// TIA Portal V16 export
// export: Created 2024-09-05T17:39:23.0698043Z, ExportSetting WithDefaults, DisplayName Totally Integrated Automation Portal, DisplayVersion V16 Update 6, DisplayName TIA Portal Version Control Interface, DisplayVersion V16 Update 2, DisplayName TIA Portal Openness, DisplayVersion V16 Update 6, DisplayName STEP 7 Professional, DisplayVersion V16 Update 6, DisplayName STEP 7 Safety, DisplayVersion V16, DisplayName WinCC Advanced, DisplayVersion V16 Update 6
FUNCTION "FC_CONFIG_MSG_IJC" : Void   // FC2, LAD
{ S7_Optimized_Access := 'TRUE' }
VERSION : 0.1
// stored: AutoNumber true, IsIECCheckEnabled false, SetENOAutomatically false, UDAEnableTagReadback false
   VAR_TEMP
      STRING_USER1 : String;
      STRING_USER2 : String;
      STRING_CORDON_1 : String;
      INDEX_IJC_CORDON : Int;
      STRING_CORDONES : Array[0..13] of String;
   END_VAR
   VAR_TEMP   // added for the SCL form of the ladder/FBD networks
      _w1 : Bool;
      _w2 : Bool;
   END_VAR
BEGIN

REGION Network 1: INDEX MSG CONFIG
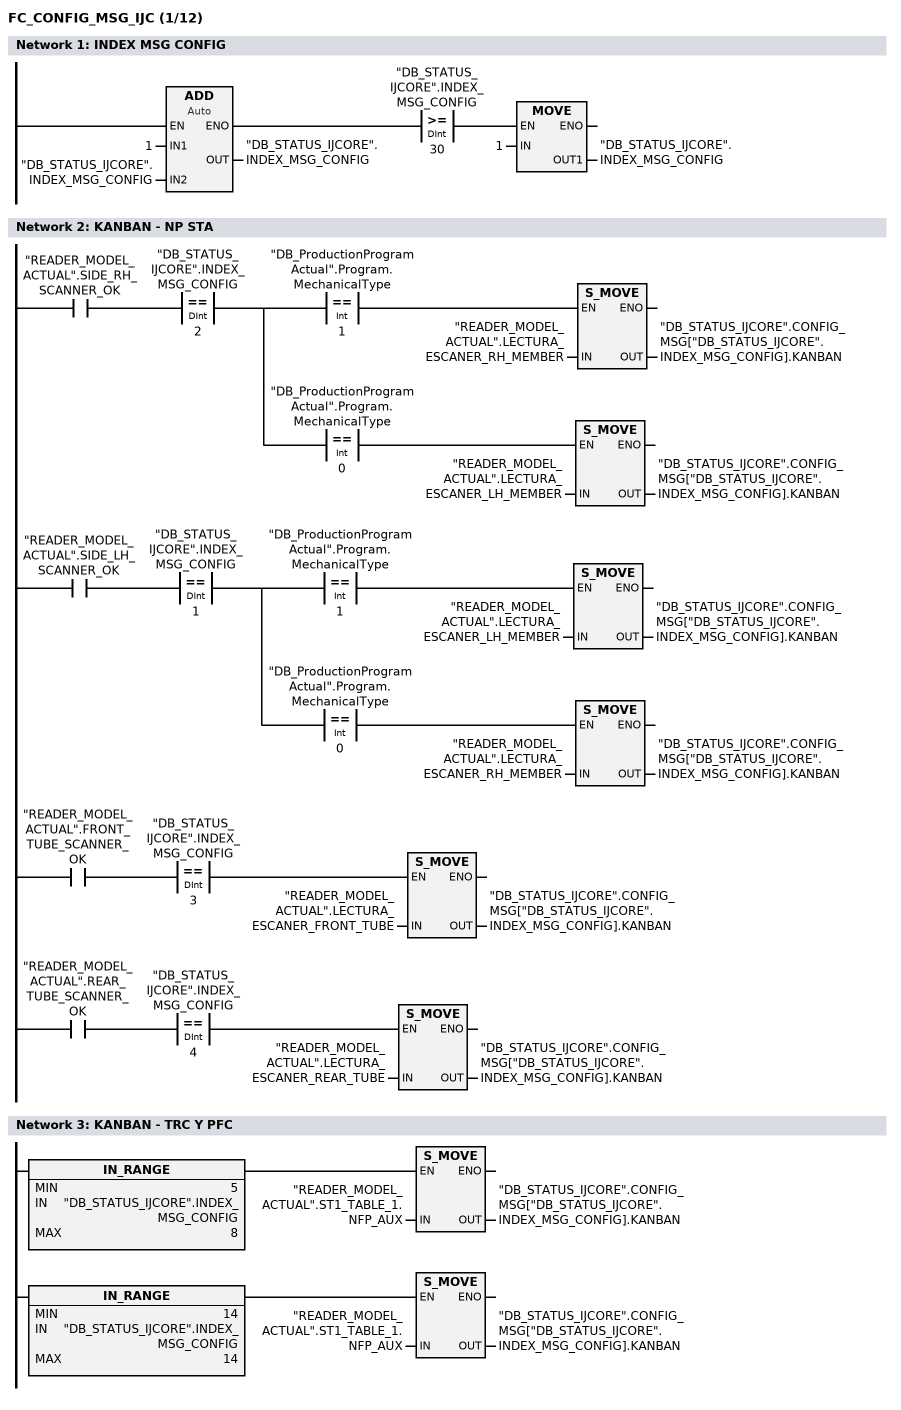
   RUNG wire#powerrail
      Add(in1 := 1, in2 := "DB_STATUS_IJCORE".INDEX_MSG_CONFIG, out => "DB_STATUS_IJCORE".INDEX_MSG_CONFIG)
      { S7_Templates := "SrcType := DInt" } GE_Contact(in1 := "DB_STATUS_IJCORE".INDEX_MSG_CONFIG, in2 := 30)
      Move(in := 1, out1 => "DB_STATUS_IJCORE".INDEX_MSG_CONFIG)
   END_RUNG
   // the same network as SCL:
   "DB_STATUS_IJCORE".INDEX_MSG_CONFIG := 1 + "DB_STATUS_IJCORE".INDEX_MSG_CONFIG;
   IF "DB_STATUS_IJCORE".INDEX_MSG_CONFIG >= 30 THEN "DB_STATUS_IJCORE".INDEX_MSG_CONFIG := 1; END_IF;
END_REGION

REGION Network 2: KANBAN - NP STA
   RUNG wire#powerrail
      Contact( "READER_MODEL_ACTUAL".SIDE_RH_SCANNER_OK )
      { S7_Templates := "SrcType := DInt" } EQ_Contact(in1 := "DB_STATUS_IJCORE".INDEX_MSG_CONFIG, in2 := 2)
      wire#w1
      { S7_Templates := "SrcType := Int" } EQ_Contact(in1 := "DB_ProductionProgramActual".Program.MechanicalType, in2 := 1)
      S_Move(in := "READER_MODEL_ACTUAL".LECTURA_ESCANER_RH_MEMBER, out => "DB_STATUS_IJCORE".CONFIG_MSG["DB_STATUS_IJCORE".INDEX_MSG_CONFIG].KANBAN)
   END_RUNG
   RUNG wire#w1
      { S7_Templates := "SrcType := Int" } EQ_Contact(in1 := "DB_ProductionProgramActual".Program.MechanicalType, in2 := 0)
      S_Move(in := "READER_MODEL_ACTUAL".LECTURA_ESCANER_LH_MEMBER, out => "DB_STATUS_IJCORE".CONFIG_MSG["DB_STATUS_IJCORE".INDEX_MSG_CONFIG].KANBAN)
   END_RUNG
   RUNG wire#powerrail
      Contact( "READER_MODEL_ACTUAL".SIDE_LH_SCANNER_OK )
      { S7_Templates := "SrcType := DInt" } EQ_Contact(in1 := "DB_STATUS_IJCORE".INDEX_MSG_CONFIG, in2 := 1)
      wire#w2
      { S7_Templates := "SrcType := Int" } EQ_Contact(in1 := "DB_ProductionProgramActual".Program.MechanicalType, in2 := 1)
      S_Move(in := "READER_MODEL_ACTUAL".LECTURA_ESCANER_LH_MEMBER, out => "DB_STATUS_IJCORE".CONFIG_MSG["DB_STATUS_IJCORE".INDEX_MSG_CONFIG].KANBAN)
   END_RUNG
   RUNG wire#w2
      { S7_Templates := "SrcType := Int" } EQ_Contact(in1 := "DB_ProductionProgramActual".Program.MechanicalType, in2 := 0)
      S_Move(in := "READER_MODEL_ACTUAL".LECTURA_ESCANER_RH_MEMBER, out => "DB_STATUS_IJCORE".CONFIG_MSG["DB_STATUS_IJCORE".INDEX_MSG_CONFIG].KANBAN)
   END_RUNG
   RUNG wire#powerrail
      Contact( "READER_MODEL_ACTUAL".FRONT_TUBE_SCANNER_OK )
      { S7_Templates := "SrcType := DInt" } EQ_Contact(in1 := "DB_STATUS_IJCORE".INDEX_MSG_CONFIG, in2 := 3)
      S_Move(in := "READER_MODEL_ACTUAL".LECTURA_ESCANER_FRONT_TUBE, out => "DB_STATUS_IJCORE".CONFIG_MSG["DB_STATUS_IJCORE".INDEX_MSG_CONFIG].KANBAN)
   END_RUNG
   RUNG wire#powerrail
      Contact( "READER_MODEL_ACTUAL".REAR_TUBE_SCANNER_OK )
      { S7_Templates := "SrcType := DInt" } EQ_Contact(in1 := "DB_STATUS_IJCORE".INDEX_MSG_CONFIG, in2 := 4)
      S_Move(in := "READER_MODEL_ACTUAL".LECTURA_ESCANER_REAR_TUBE, out => "DB_STATUS_IJCORE".CONFIG_MSG["DB_STATUS_IJCORE".INDEX_MSG_CONFIG].KANBAN)
   END_RUNG
   // the same network as SCL:
   #_w1 := "READER_MODEL_ACTUAL".SIDE_RH_SCANNER_OK AND ("DB_STATUS_IJCORE".INDEX_MSG_CONFIG = 2);
   IF #_w1 AND ("DB_ProductionProgramActual".Program.MechanicalType = 1) THEN
       "DB_STATUS_IJCORE".CONFIG_MSG["DB_STATUS_IJCORE".INDEX_MSG_CONFIG].KANBAN := "READER_MODEL_ACTUAL".LECTURA_ESCANER_RH_MEMBER;
   END_IF;
   IF #_w1 AND ("DB_ProductionProgramActual".Program.MechanicalType = 0) THEN
       "DB_STATUS_IJCORE".CONFIG_MSG["DB_STATUS_IJCORE".INDEX_MSG_CONFIG].KANBAN := "READER_MODEL_ACTUAL".LECTURA_ESCANER_LH_MEMBER;
   END_IF;
   #_w2 := "READER_MODEL_ACTUAL".SIDE_LH_SCANNER_OK AND ("DB_STATUS_IJCORE".INDEX_MSG_CONFIG = 1);
   IF #_w2 AND ("DB_ProductionProgramActual".Program.MechanicalType = 1) THEN
       "DB_STATUS_IJCORE".CONFIG_MSG["DB_STATUS_IJCORE".INDEX_MSG_CONFIG].KANBAN := "READER_MODEL_ACTUAL".LECTURA_ESCANER_LH_MEMBER;
   END_IF;
   IF #_w2 AND ("DB_ProductionProgramActual".Program.MechanicalType = 0) THEN
       "DB_STATUS_IJCORE".CONFIG_MSG["DB_STATUS_IJCORE".INDEX_MSG_CONFIG].KANBAN := "READER_MODEL_ACTUAL".LECTURA_ESCANER_RH_MEMBER;
   END_IF;
   IF "READER_MODEL_ACTUAL".FRONT_TUBE_SCANNER_OK AND ("DB_STATUS_IJCORE".INDEX_MSG_CONFIG = 3) THEN
       "DB_STATUS_IJCORE".CONFIG_MSG["DB_STATUS_IJCORE".INDEX_MSG_CONFIG].KANBAN := "READER_MODEL_ACTUAL".LECTURA_ESCANER_FRONT_TUBE;
   END_IF;
   IF "READER_MODEL_ACTUAL".REAR_TUBE_SCANNER_OK AND ("DB_STATUS_IJCORE".INDEX_MSG_CONFIG = 4) THEN
       "DB_STATUS_IJCORE".CONFIG_MSG["DB_STATUS_IJCORE".INDEX_MSG_CONFIG].KANBAN := "READER_MODEL_ACTUAL".LECTURA_ESCANER_REAR_TUBE;
   END_IF;
END_REGION

REGION Network 3: KANBAN - TRC Y PFC
   RUNG wire#powerrail
      { S7_Templates := "SrcType := DInt" } InRange(min := 5, in := "DB_STATUS_IJCORE".INDEX_MSG_CONFIG, max := 8)
      S_Move(in := "READER_MODEL_ACTUAL".ST1_TABLE_1.NFP_AUX, out => "DB_STATUS_IJCORE".CONFIG_MSG["DB_STATUS_IJCORE".INDEX_MSG_CONFIG].KANBAN)
   END_RUNG
   RUNG wire#powerrail
      { S7_Templates := "SrcType := DInt" } InRange(min := 14, in := "DB_STATUS_IJCORE".INDEX_MSG_CONFIG, max := 14)
      S_Move(in := "READER_MODEL_ACTUAL".ST1_TABLE_1.NFP_AUX, out => "DB_STATUS_IJCORE".CONFIG_MSG["DB_STATUS_IJCORE".INDEX_MSG_CONFIG].KANBAN)
   END_RUNG
   // the same network as SCL:
   IF (5 <= "DB_STATUS_IJCORE".INDEX_MSG_CONFIG) AND ("DB_STATUS_IJCORE".INDEX_MSG_CONFIG <= 8) THEN
       "DB_STATUS_IJCORE".CONFIG_MSG["DB_STATUS_IJCORE".INDEX_MSG_CONFIG].KANBAN := "READER_MODEL_ACTUAL".ST1_TABLE_1.NFP_AUX;
   END_IF;
   IF (14 <= "DB_STATUS_IJCORE".INDEX_MSG_CONFIG) AND ("DB_STATUS_IJCORE".INDEX_MSG_CONFIG <= 14) THEN
       "DB_STATUS_IJCORE".CONFIG_MSG["DB_STATUS_IJCORE".INDEX_MSG_CONFIG].KANBAN := "READER_MODEL_ACTUAL".ST1_TABLE_1.NFP_AUX;
   END_IF;
END_REGION

REGION Network 4: KANBAN - TRR Y CNF
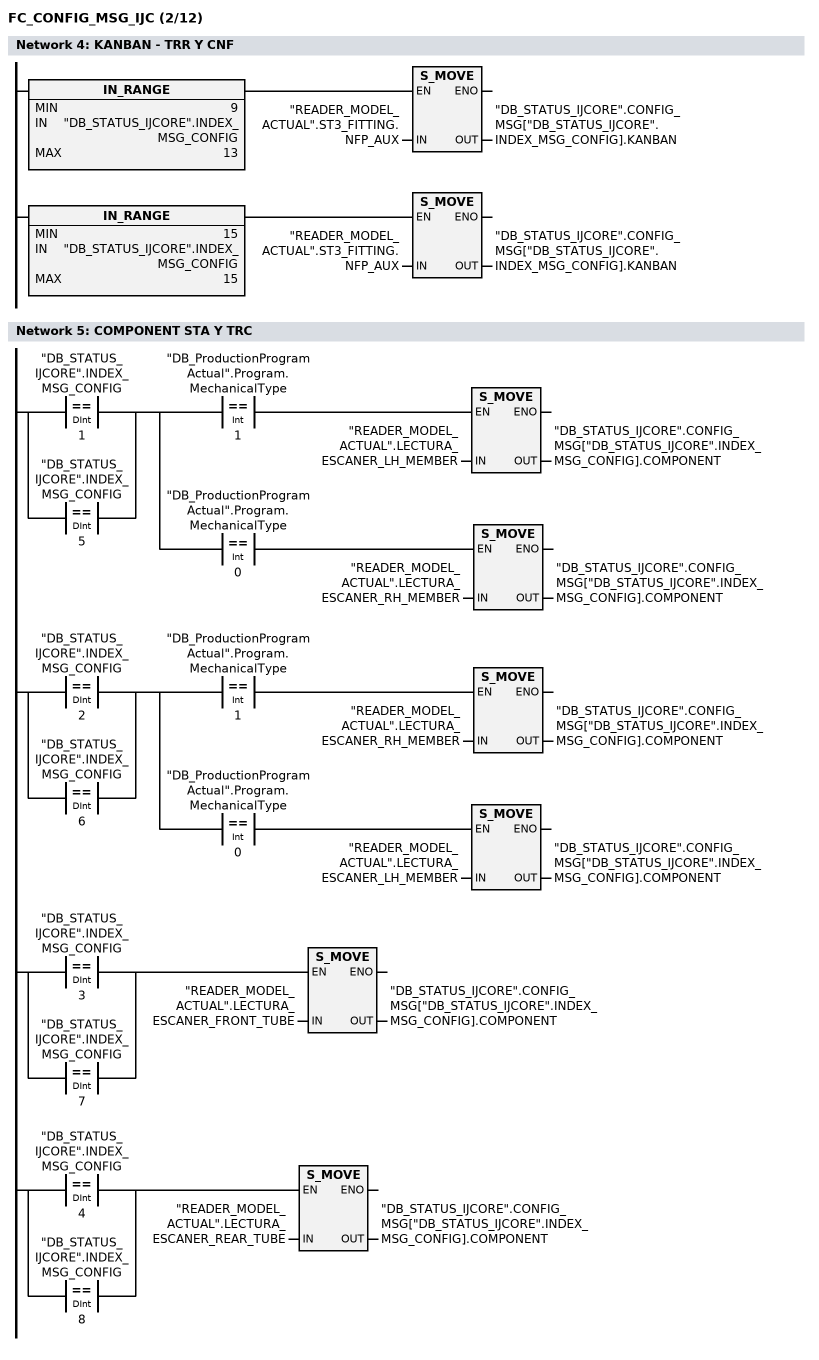
   RUNG wire#powerrail
      { S7_Templates := "SrcType := DInt" } InRange(min := 9, in := "DB_STATUS_IJCORE".INDEX_MSG_CONFIG, max := 13)
      S_Move(in := "READER_MODEL_ACTUAL".ST3_FITTING.NFP_AUX, out => "DB_STATUS_IJCORE".CONFIG_MSG["DB_STATUS_IJCORE".INDEX_MSG_CONFIG].KANBAN)
   END_RUNG
   RUNG wire#powerrail
      { S7_Templates := "SrcType := DInt" } InRange(min := 15, in := "DB_STATUS_IJCORE".INDEX_MSG_CONFIG, max := 15)
      S_Move(in := "READER_MODEL_ACTUAL".ST3_FITTING.NFP_AUX, out => "DB_STATUS_IJCORE".CONFIG_MSG["DB_STATUS_IJCORE".INDEX_MSG_CONFIG].KANBAN)
   END_RUNG
   // the same network as SCL:
   IF (9 <= "DB_STATUS_IJCORE".INDEX_MSG_CONFIG) AND ("DB_STATUS_IJCORE".INDEX_MSG_CONFIG <= 13) THEN
       "DB_STATUS_IJCORE".CONFIG_MSG["DB_STATUS_IJCORE".INDEX_MSG_CONFIG].KANBAN := "READER_MODEL_ACTUAL".ST3_FITTING.NFP_AUX;
   END_IF;
   IF (15 <= "DB_STATUS_IJCORE".INDEX_MSG_CONFIG) AND ("DB_STATUS_IJCORE".INDEX_MSG_CONFIG <= 15) THEN
       "DB_STATUS_IJCORE".CONFIG_MSG["DB_STATUS_IJCORE".INDEX_MSG_CONFIG].KANBAN := "READER_MODEL_ACTUAL".ST3_FITTING.NFP_AUX;
   END_IF;
END_REGION

REGION Network 5: COMPONENT STA Y TRC
   RUNG wire#powerrail
      { S7_Templates := "SrcType := DInt" } EQ_Contact(in1 := "DB_STATUS_IJCORE".INDEX_MSG_CONFIG, in2 := 1)
      wire#w1
      { S7_Templates := "SrcType := Int" } EQ_Contact(in1 := "DB_ProductionProgramActual".Program.MechanicalType, in2 := 1)
      S_Move(in := "READER_MODEL_ACTUAL".LECTURA_ESCANER_LH_MEMBER, out => "DB_STATUS_IJCORE".CONFIG_MSG["DB_STATUS_IJCORE".INDEX_MSG_CONFIG].COMPONENT)
   END_RUNG
   RUNG wire#powerrail
      { S7_Templates := "SrcType := DInt" } EQ_Contact(in1 := "DB_STATUS_IJCORE".INDEX_MSG_CONFIG, in2 := 5)
   END_RUNG wire#w1
   RUNG wire#w1
      { S7_Templates := "SrcType := Int" } EQ_Contact(in1 := "DB_ProductionProgramActual".Program.MechanicalType, in2 := 0)
      S_Move(in := "READER_MODEL_ACTUAL".LECTURA_ESCANER_RH_MEMBER, out => "DB_STATUS_IJCORE".CONFIG_MSG["DB_STATUS_IJCORE".INDEX_MSG_CONFIG].COMPONENT)
   END_RUNG
   RUNG wire#powerrail
      { S7_Templates := "SrcType := DInt" } EQ_Contact(in1 := "DB_STATUS_IJCORE".INDEX_MSG_CONFIG, in2 := 2)
      wire#w2
      { S7_Templates := "SrcType := Int" } EQ_Contact(in1 := "DB_ProductionProgramActual".Program.MechanicalType, in2 := 1)
      S_Move(in := "READER_MODEL_ACTUAL".LECTURA_ESCANER_RH_MEMBER, out => "DB_STATUS_IJCORE".CONFIG_MSG["DB_STATUS_IJCORE".INDEX_MSG_CONFIG].COMPONENT)
   END_RUNG
   RUNG wire#powerrail
      { S7_Templates := "SrcType := DInt" } EQ_Contact(in1 := "DB_STATUS_IJCORE".INDEX_MSG_CONFIG, in2 := 6)
   END_RUNG wire#w2
   RUNG wire#w2
      { S7_Templates := "SrcType := Int" } EQ_Contact(in1 := "DB_ProductionProgramActual".Program.MechanicalType, in2 := 0)
      S_Move(in := "READER_MODEL_ACTUAL".LECTURA_ESCANER_LH_MEMBER, out => "DB_STATUS_IJCORE".CONFIG_MSG["DB_STATUS_IJCORE".INDEX_MSG_CONFIG].COMPONENT)
   END_RUNG
   RUNG wire#powerrail
      { S7_Templates := "SrcType := DInt" } EQ_Contact(in1 := "DB_STATUS_IJCORE".INDEX_MSG_CONFIG, in2 := 3)
      wire#w3
      S_Move(in := "READER_MODEL_ACTUAL".LECTURA_ESCANER_FRONT_TUBE, out => "DB_STATUS_IJCORE".CONFIG_MSG["DB_STATUS_IJCORE".INDEX_MSG_CONFIG].COMPONENT)
   END_RUNG
   RUNG wire#powerrail
      { S7_Templates := "SrcType := DInt" } EQ_Contact(in1 := "DB_STATUS_IJCORE".INDEX_MSG_CONFIG, in2 := 7)
   END_RUNG wire#w3
   RUNG wire#powerrail
      { S7_Templates := "SrcType := DInt" } EQ_Contact(in1 := "DB_STATUS_IJCORE".INDEX_MSG_CONFIG, in2 := 4)
      wire#w4
      S_Move(in := "READER_MODEL_ACTUAL".LECTURA_ESCANER_REAR_TUBE, out => "DB_STATUS_IJCORE".CONFIG_MSG["DB_STATUS_IJCORE".INDEX_MSG_CONFIG].COMPONENT)
   END_RUNG
   RUNG wire#powerrail
      { S7_Templates := "SrcType := DInt" } EQ_Contact(in1 := "DB_STATUS_IJCORE".INDEX_MSG_CONFIG, in2 := 8)
   END_RUNG wire#w4
   // the same network as SCL:
   #_w1 := ("DB_STATUS_IJCORE".INDEX_MSG_CONFIG = 1) OR ("DB_STATUS_IJCORE".INDEX_MSG_CONFIG = 5);
   IF #_w1 AND ("DB_ProductionProgramActual".Program.MechanicalType = 1) THEN
       "DB_STATUS_IJCORE".CONFIG_MSG["DB_STATUS_IJCORE".INDEX_MSG_CONFIG].COMPONENT := "READER_MODEL_ACTUAL".LECTURA_ESCANER_LH_MEMBER;
   END_IF;
   IF #_w1 AND ("DB_ProductionProgramActual".Program.MechanicalType = 0) THEN
       "DB_STATUS_IJCORE".CONFIG_MSG["DB_STATUS_IJCORE".INDEX_MSG_CONFIG].COMPONENT := "READER_MODEL_ACTUAL".LECTURA_ESCANER_RH_MEMBER;
   END_IF;
   #_w2 := ("DB_STATUS_IJCORE".INDEX_MSG_CONFIG = 2) OR ("DB_STATUS_IJCORE".INDEX_MSG_CONFIG = 6);
   IF #_w2 AND ("DB_ProductionProgramActual".Program.MechanicalType = 1) THEN
       "DB_STATUS_IJCORE".CONFIG_MSG["DB_STATUS_IJCORE".INDEX_MSG_CONFIG].COMPONENT := "READER_MODEL_ACTUAL".LECTURA_ESCANER_RH_MEMBER;
   END_IF;
   IF #_w2 AND ("DB_ProductionProgramActual".Program.MechanicalType = 0) THEN
       "DB_STATUS_IJCORE".CONFIG_MSG["DB_STATUS_IJCORE".INDEX_MSG_CONFIG].COMPONENT := "READER_MODEL_ACTUAL".LECTURA_ESCANER_LH_MEMBER;
   END_IF;
   IF ("DB_STATUS_IJCORE".INDEX_MSG_CONFIG = 3) OR ("DB_STATUS_IJCORE".INDEX_MSG_CONFIG = 7) THEN
       "DB_STATUS_IJCORE".CONFIG_MSG["DB_STATUS_IJCORE".INDEX_MSG_CONFIG].COMPONENT := "READER_MODEL_ACTUAL".LECTURA_ESCANER_FRONT_TUBE;
   END_IF;
   IF ("DB_STATUS_IJCORE".INDEX_MSG_CONFIG = 4) OR ("DB_STATUS_IJCORE".INDEX_MSG_CONFIG = 8) THEN
       "DB_STATUS_IJCORE".CONFIG_MSG["DB_STATUS_IJCORE".INDEX_MSG_CONFIG].COMPONENT := "READER_MODEL_ACTUAL".LECTURA_ESCANER_REAR_TUBE;
   END_IF;
END_REGION

REGION Network 6: COMPONENT PFC
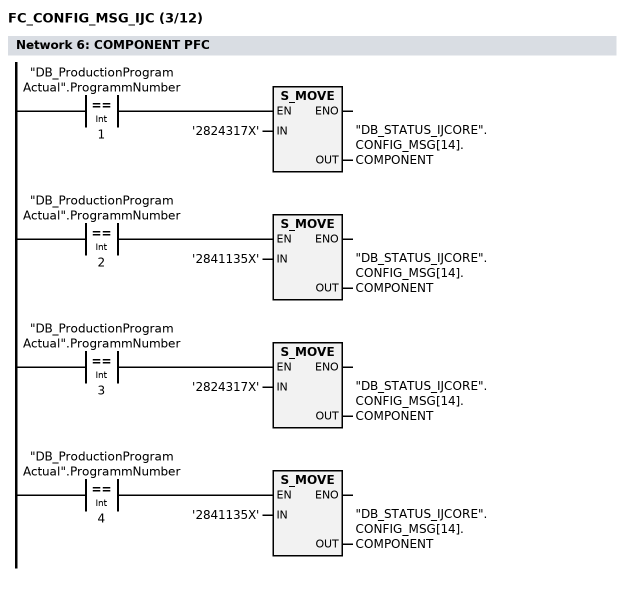
   RUNG wire#powerrail
      { S7_Templates := "SrcType := Int" } EQ_Contact(in1 := "DB_ProductionProgramActual".ProgrammNumber, in2 := 1)
      S_Move(in := '2824317X', out => "DB_STATUS_IJCORE".CONFIG_MSG[14].COMPONENT)
   END_RUNG
   RUNG wire#powerrail
      { S7_Templates := "SrcType := Int" } EQ_Contact(in1 := "DB_ProductionProgramActual".ProgrammNumber, in2 := 2)
      S_Move(in := '2841135X', out => "DB_STATUS_IJCORE".CONFIG_MSG[14].COMPONENT)
   END_RUNG
   RUNG wire#powerrail
      { S7_Templates := "SrcType := Int" } EQ_Contact(in1 := "DB_ProductionProgramActual".ProgrammNumber, in2 := 3)
      S_Move(in := '2824317X', out => "DB_STATUS_IJCORE".CONFIG_MSG[14].COMPONENT)
   END_RUNG
   RUNG wire#powerrail
      { S7_Templates := "SrcType := Int" } EQ_Contact(in1 := "DB_ProductionProgramActual".ProgrammNumber, in2 := 4)
      S_Move(in := '2841135X', out => "DB_STATUS_IJCORE".CONFIG_MSG[14].COMPONENT)
   END_RUNG
   // the same network as SCL:
   IF "DB_ProductionProgramActual".ProgrammNumber = 1 THEN
       "DB_STATUS_IJCORE".CONFIG_MSG[14].COMPONENT := '2824317X';
   END_IF;
   IF "DB_ProductionProgramActual".ProgrammNumber = 2 THEN
       "DB_STATUS_IJCORE".CONFIG_MSG[14].COMPONENT := '2841135X';
   END_IF;
   IF "DB_ProductionProgramActual".ProgrammNumber = 3 THEN
       "DB_STATUS_IJCORE".CONFIG_MSG[14].COMPONENT := '2824317X';
   END_IF;
   IF "DB_ProductionProgramActual".ProgrammNumber = 4 THEN
       "DB_STATUS_IJCORE".CONFIG_MSG[14].COMPONENT := '2841135X';
   END_IF;
END_REGION

REGION Network 7: COMPONENT CNF
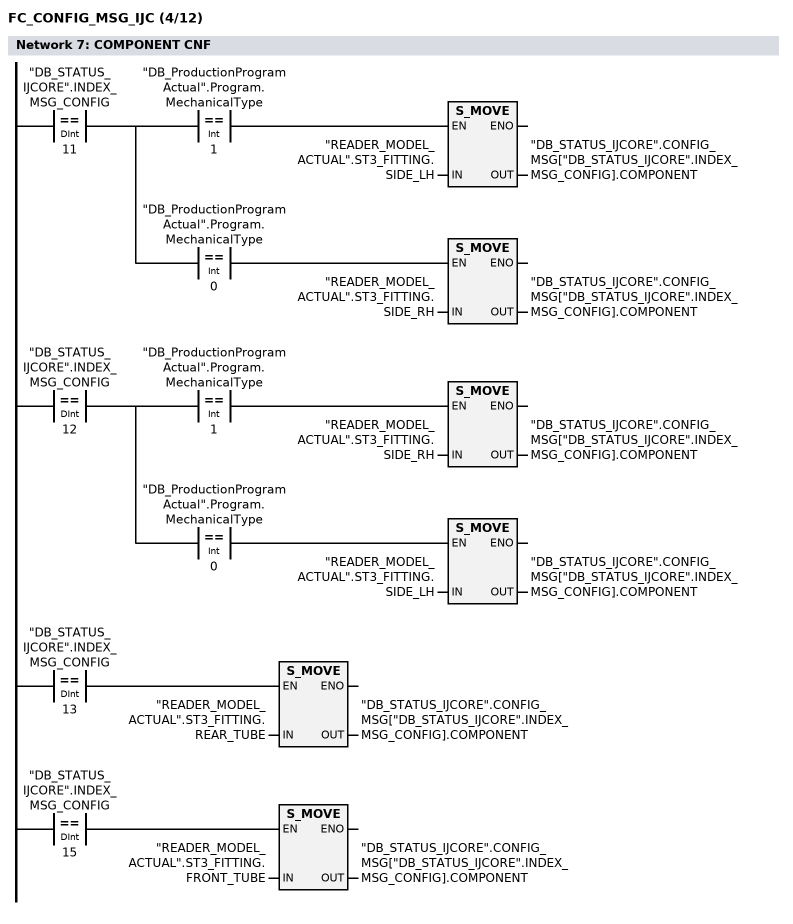
   RUNG wire#powerrail
      { S7_Templates := "SrcType := DInt" } EQ_Contact(in1 := "DB_STATUS_IJCORE".INDEX_MSG_CONFIG, in2 := 11)
      wire#w1
      { S7_Templates := "SrcType := Int" } EQ_Contact(in1 := "DB_ProductionProgramActual".Program.MechanicalType, in2 := 1)
      S_Move(in := "READER_MODEL_ACTUAL".ST3_FITTING.SIDE_LH, out => "DB_STATUS_IJCORE".CONFIG_MSG["DB_STATUS_IJCORE".INDEX_MSG_CONFIG].COMPONENT)
   END_RUNG
   RUNG wire#w1
      { S7_Templates := "SrcType := Int" } EQ_Contact(in1 := "DB_ProductionProgramActual".Program.MechanicalType, in2 := 0)
      S_Move(in := "READER_MODEL_ACTUAL".ST3_FITTING.SIDE_RH, out => "DB_STATUS_IJCORE".CONFIG_MSG["DB_STATUS_IJCORE".INDEX_MSG_CONFIG].COMPONENT)
   END_RUNG
   RUNG wire#powerrail
      { S7_Templates := "SrcType := DInt" } EQ_Contact(in1 := "DB_STATUS_IJCORE".INDEX_MSG_CONFIG, in2 := 12)
      wire#w2
      { S7_Templates := "SrcType := Int" } EQ_Contact(in1 := "DB_ProductionProgramActual".Program.MechanicalType, in2 := 1)
      S_Move(in := "READER_MODEL_ACTUAL".ST3_FITTING.SIDE_RH, out => "DB_STATUS_IJCORE".CONFIG_MSG["DB_STATUS_IJCORE".INDEX_MSG_CONFIG].COMPONENT)
   END_RUNG
   RUNG wire#w2
      { S7_Templates := "SrcType := Int" } EQ_Contact(in1 := "DB_ProductionProgramActual".Program.MechanicalType, in2 := 0)
      S_Move(in := "READER_MODEL_ACTUAL".ST3_FITTING.SIDE_LH, out => "DB_STATUS_IJCORE".CONFIG_MSG["DB_STATUS_IJCORE".INDEX_MSG_CONFIG].COMPONENT)
   END_RUNG
   RUNG wire#powerrail
      { S7_Templates := "SrcType := DInt" } EQ_Contact(in1 := "DB_STATUS_IJCORE".INDEX_MSG_CONFIG, in2 := 13)
      S_Move(in := "READER_MODEL_ACTUAL".ST3_FITTING.REAR_TUBE, out => "DB_STATUS_IJCORE".CONFIG_MSG["DB_STATUS_IJCORE".INDEX_MSG_CONFIG].COMPONENT)
   END_RUNG
   RUNG wire#powerrail
      { S7_Templates := "SrcType := DInt" } EQ_Contact(in1 := "DB_STATUS_IJCORE".INDEX_MSG_CONFIG, in2 := 15)
      S_Move(in := "READER_MODEL_ACTUAL".ST3_FITTING.FRONT_TUBE, out => "DB_STATUS_IJCORE".CONFIG_MSG["DB_STATUS_IJCORE".INDEX_MSG_CONFIG].COMPONENT)
   END_RUNG
   // the same network as SCL:
   #_w1 := "DB_STATUS_IJCORE".INDEX_MSG_CONFIG = 11;
   IF #_w1 AND ("DB_ProductionProgramActual".Program.MechanicalType = 1) THEN
       "DB_STATUS_IJCORE".CONFIG_MSG["DB_STATUS_IJCORE".INDEX_MSG_CONFIG].COMPONENT := "READER_MODEL_ACTUAL".ST3_FITTING.SIDE_LH;
   END_IF;
   IF #_w1 AND ("DB_ProductionProgramActual".Program.MechanicalType = 0) THEN
       "DB_STATUS_IJCORE".CONFIG_MSG["DB_STATUS_IJCORE".INDEX_MSG_CONFIG].COMPONENT := "READER_MODEL_ACTUAL".ST3_FITTING.SIDE_RH;
   END_IF;
   #_w2 := "DB_STATUS_IJCORE".INDEX_MSG_CONFIG = 12;
   IF #_w2 AND ("DB_ProductionProgramActual".Program.MechanicalType = 1) THEN
       "DB_STATUS_IJCORE".CONFIG_MSG["DB_STATUS_IJCORE".INDEX_MSG_CONFIG].COMPONENT := "READER_MODEL_ACTUAL".ST3_FITTING.SIDE_RH;
   END_IF;
   IF #_w2 AND ("DB_ProductionProgramActual".Program.MechanicalType = 0) THEN
       "DB_STATUS_IJCORE".CONFIG_MSG["DB_STATUS_IJCORE".INDEX_MSG_CONFIG].COMPONENT := "READER_MODEL_ACTUAL".ST3_FITTING.SIDE_LH;
   END_IF;
   IF "DB_STATUS_IJCORE".INDEX_MSG_CONFIG = 13 THEN
       "DB_STATUS_IJCORE".CONFIG_MSG["DB_STATUS_IJCORE".INDEX_MSG_CONFIG].COMPONENT := "READER_MODEL_ACTUAL".ST3_FITTING.REAR_TUBE;
   END_IF;
   IF "DB_STATUS_IJCORE".INDEX_MSG_CONFIG = 15 THEN
       "DB_STATUS_IJCORE".CONFIG_MSG["DB_STATUS_IJCORE".INDEX_MSG_CONFIG].COMPONENT := "READER_MODEL_ACTUAL".ST3_FITTING.FRONT_TUBE;
   END_IF;
END_REGION

REGION Network 8: STATUS TRR
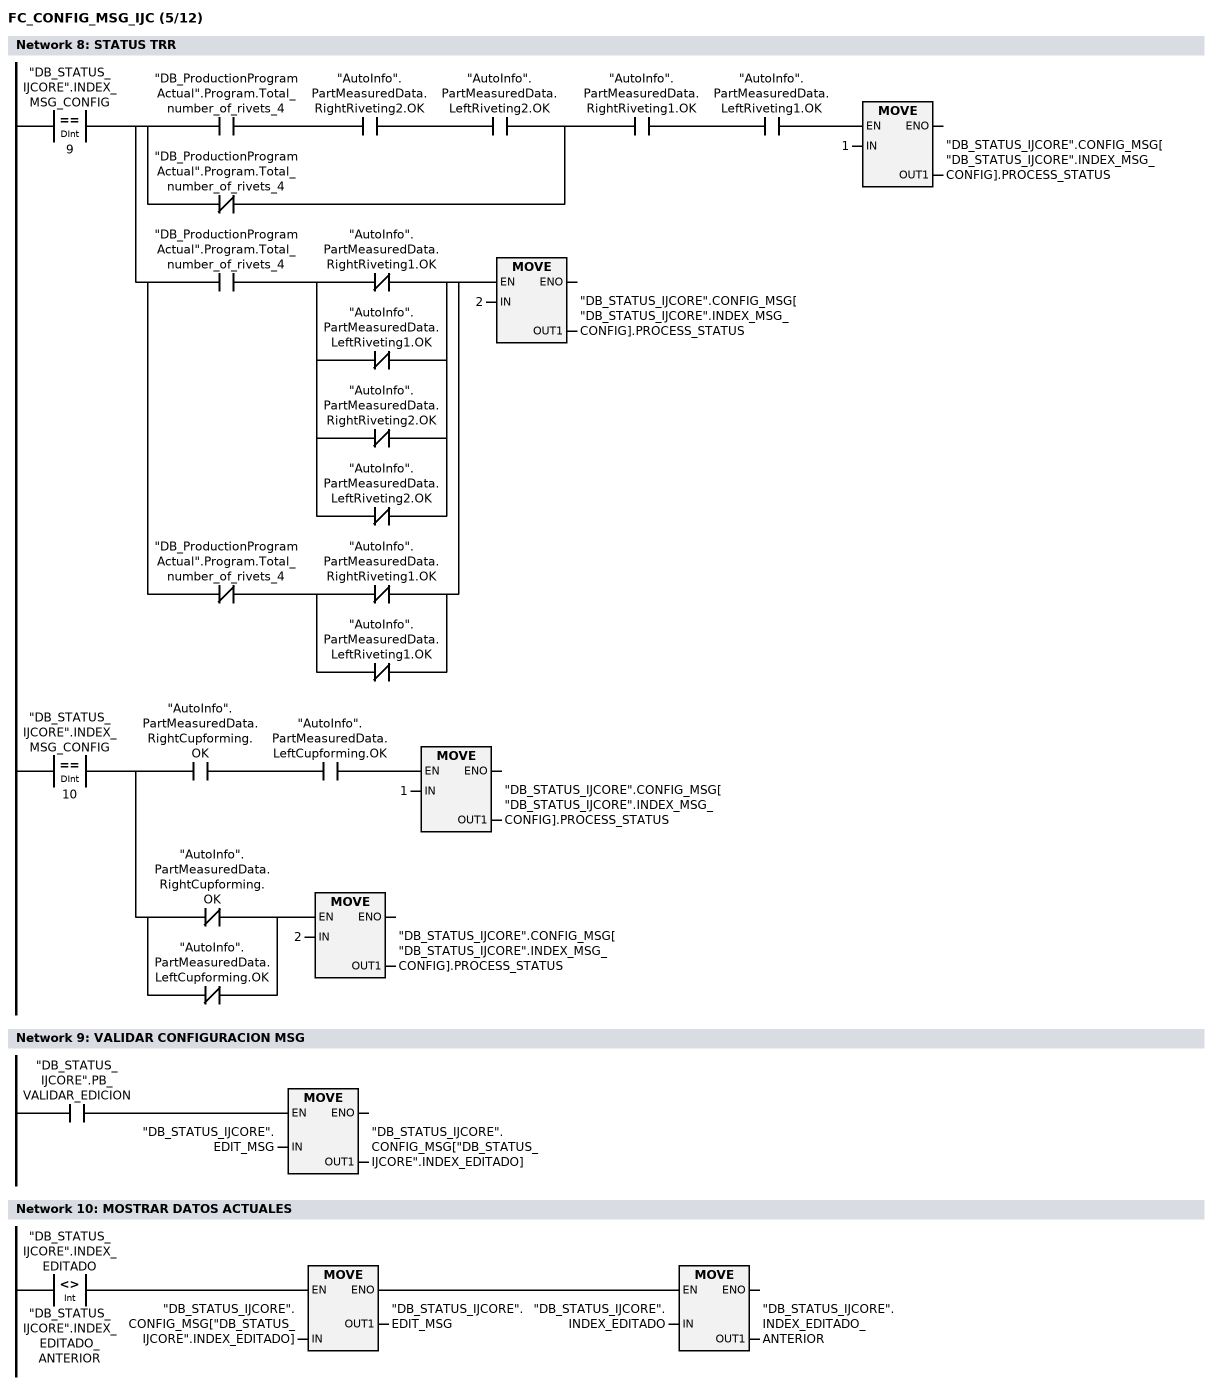
   RUNG wire#powerrail
      { S7_Templates := "SrcType := DInt" } EQ_Contact(in1 := "DB_STATUS_IJCORE".INDEX_MSG_CONFIG, in2 := 9)
      wire#w1
      Contact( "DB_ProductionProgramActual".Program.Total_number_of_rivets_4 )
      Contact( "AutoInfo".PartMeasuredData.RightRiveting2.OK )
      Contact( "AutoInfo".PartMeasuredData.LeftRiveting2.OK )
      wire#w2
      Contact( "AutoInfo".PartMeasuredData.RightRiveting1.OK )
      Contact( "AutoInfo".PartMeasuredData.LeftRiveting1.OK )
      Move(in := 1, out1 => "DB_STATUS_IJCORE".CONFIG_MSG["DB_STATUS_IJCORE".INDEX_MSG_CONFIG].PROCESS_STATUS)
   END_RUNG
   RUNG wire#w1
      I_Contact( "DB_ProductionProgramActual".Program.Total_number_of_rivets_4 )
   END_RUNG wire#w2
   RUNG wire#w1
      Contact( "DB_ProductionProgramActual".Program.Total_number_of_rivets_4 )
      wire#w3
      I_Contact( "AutoInfo".PartMeasuredData.RightRiveting1.OK )
      wire#w4
      Move(in := 2, out1 => "DB_STATUS_IJCORE".CONFIG_MSG["DB_STATUS_IJCORE".INDEX_MSG_CONFIG].PROCESS_STATUS)
   END_RUNG
   RUNG wire#w3
      I_Contact( "AutoInfo".PartMeasuredData.LeftRiveting1.OK )
   END_RUNG wire#w4
   RUNG wire#w3
      I_Contact( "AutoInfo".PartMeasuredData.RightRiveting2.OK )
   END_RUNG wire#w4
   RUNG wire#w3
      I_Contact( "AutoInfo".PartMeasuredData.LeftRiveting2.OK )
   END_RUNG wire#w4
   RUNG wire#w1
      I_Contact( "DB_ProductionProgramActual".Program.Total_number_of_rivets_4 )
      wire#w5
      I_Contact( "AutoInfo".PartMeasuredData.RightRiveting1.OK )
   END_RUNG wire#w4
   RUNG wire#w5
      I_Contact( "AutoInfo".PartMeasuredData.LeftRiveting1.OK )
   END_RUNG wire#w4
   RUNG wire#powerrail
      { S7_Templates := "SrcType := DInt" } EQ_Contact(in1 := "DB_STATUS_IJCORE".INDEX_MSG_CONFIG, in2 := 10)
      wire#w6
      Contact( "AutoInfo".PartMeasuredData.RightCupforming.OK )
      Contact( "AutoInfo".PartMeasuredData.LeftCupforming.OK )
      Move(in := 1, out1 => "DB_STATUS_IJCORE".CONFIG_MSG["DB_STATUS_IJCORE".INDEX_MSG_CONFIG].PROCESS_STATUS)
   END_RUNG
   RUNG wire#w6
      I_Contact( "AutoInfo".PartMeasuredData.RightCupforming.OK )
      wire#w7
      Move(in := 2, out1 => "DB_STATUS_IJCORE".CONFIG_MSG["DB_STATUS_IJCORE".INDEX_MSG_CONFIG].PROCESS_STATUS)
   END_RUNG
   RUNG wire#w6
      I_Contact( "AutoInfo".PartMeasuredData.LeftCupforming.OK )
   END_RUNG wire#w7
   // the same network as SCL:
   #_w1 := "DB_STATUS_IJCORE".INDEX_MSG_CONFIG = 9;
   IF #_w1 AND (("DB_ProductionProgramActual".Program.Total_number_of_rivets_4 AND "AutoInfo".PartMeasuredData.RightRiveting2.OK AND "AutoInfo".PartMeasuredData.LeftRiveting2.OK) OR NOT "DB_ProductionProgramActual".Program.Total_number_of_rivets_4) AND "AutoInfo".PartMeasuredData.RightRiveting1.OK AND "AutoInfo".PartMeasuredData.LeftRiveting1.OK THEN
       "DB_STATUS_IJCORE".CONFIG_MSG["DB_STATUS_IJCORE".INDEX_MSG_CONFIG].PROCESS_STATUS := 1;
   END_IF;
   IF #_w1 AND (("DB_ProductionProgramActual".Program.Total_number_of_rivets_4 AND (NOT "AutoInfo".PartMeasuredData.RightRiveting1.OK OR NOT "AutoInfo".PartMeasuredData.LeftRiveting1.OK OR NOT "AutoInfo".PartMeasuredData.RightRiveting2.OK OR NOT "AutoInfo".PartMeasuredData.LeftRiveting2.OK)) OR (NOT "DB_ProductionProgramActual".Program.Total_number_of_rivets_4 AND (NOT "AutoInfo".PartMeasuredData.RightRiveting1.OK OR NOT "AutoInfo".PartMeasuredData.LeftRiveting1.OK))) THEN
       "DB_STATUS_IJCORE".CONFIG_MSG["DB_STATUS_IJCORE".INDEX_MSG_CONFIG].PROCESS_STATUS := 2;
   END_IF;
   #_w2 := "DB_STATUS_IJCORE".INDEX_MSG_CONFIG = 10;
   IF #_w2 AND "AutoInfo".PartMeasuredData.RightCupforming.OK AND "AutoInfo".PartMeasuredData.LeftCupforming.OK THEN
       "DB_STATUS_IJCORE".CONFIG_MSG["DB_STATUS_IJCORE".INDEX_MSG_CONFIG].PROCESS_STATUS := 1;
   END_IF;
   IF #_w2 AND (NOT "AutoInfo".PartMeasuredData.RightCupforming.OK OR NOT "AutoInfo".PartMeasuredData.LeftCupforming.OK) THEN
       "DB_STATUS_IJCORE".CONFIG_MSG["DB_STATUS_IJCORE".INDEX_MSG_CONFIG].PROCESS_STATUS := 2;
   END_IF;
END_REGION

REGION Network 9: VALIDAR CONFIGURACION MSG
   RUNG wire#powerrail
      Contact( "DB_STATUS_IJCORE".PB_VALIDAR_EDICION )
      Move(in := "DB_STATUS_IJCORE".EDIT_MSG, out1 => "DB_STATUS_IJCORE".CONFIG_MSG["DB_STATUS_IJCORE".INDEX_EDITADO])
   END_RUNG
   // the same network as SCL:
   IF "DB_STATUS_IJCORE".PB_VALIDAR_EDICION THEN
       "DB_STATUS_IJCORE".CONFIG_MSG["DB_STATUS_IJCORE".INDEX_EDITADO] := "DB_STATUS_IJCORE".EDIT_MSG;
   END_IF;
END_REGION

REGION Network 10: MOSTRAR DATOS ACTUALES
   RUNG wire#powerrail
      { S7_Templates := "SrcType := Int" } NE_Contact(in1 := "DB_STATUS_IJCORE".INDEX_EDITADO, in2 := "DB_STATUS_IJCORE".INDEX_EDITADO_ANTERIOR)
      Move(in := "DB_STATUS_IJCORE".CONFIG_MSG["DB_STATUS_IJCORE".INDEX_EDITADO], out1 => "DB_STATUS_IJCORE".EDIT_MSG)
      Move(in := "DB_STATUS_IJCORE".INDEX_EDITADO, out1 => "DB_STATUS_IJCORE".INDEX_EDITADO_ANTERIOR)
   END_RUNG
   // the same network as SCL:
   IF "DB_STATUS_IJCORE".INDEX_EDITADO <> "DB_STATUS_IJCORE".INDEX_EDITADO_ANTERIOR THEN
       "DB_STATUS_IJCORE".EDIT_MSG := "DB_STATUS_IJCORE".CONFIG_MSG["DB_STATUS_IJCORE".INDEX_EDITADO];
       "DB_STATUS_IJCORE".INDEX_EDITADO_ANTERIOR := "DB_STATUS_IJCORE".INDEX_EDITADO;
   END_IF;
END_REGION

REGION Network 11: SEND STA
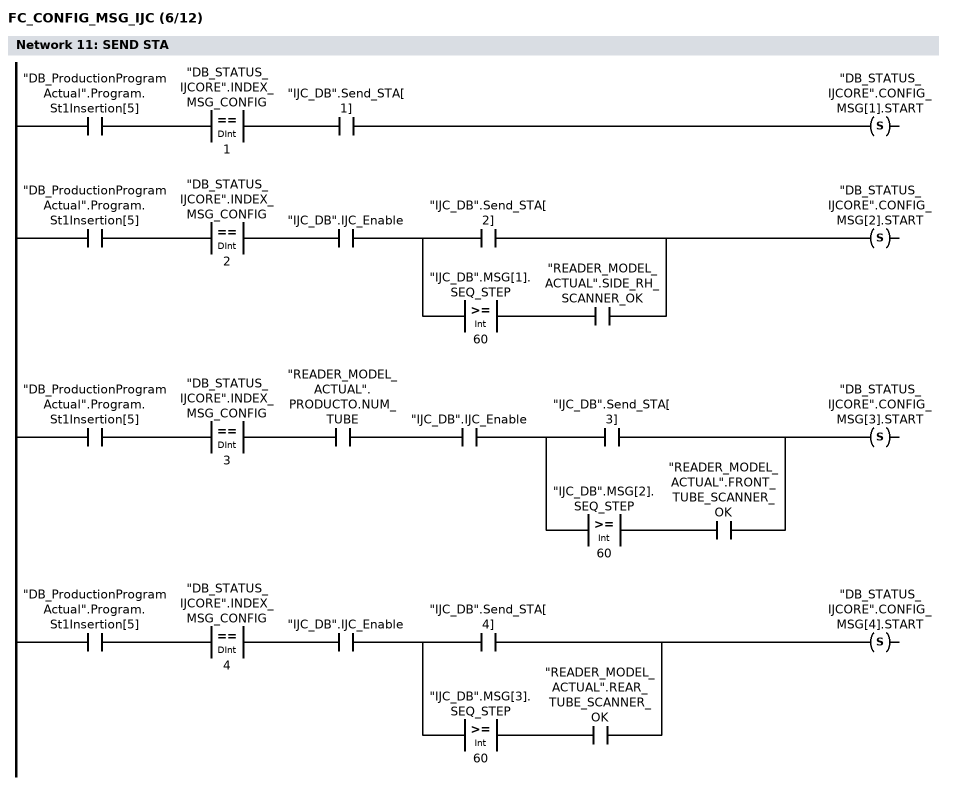
   RUNG wire#powerrail
      Contact( "DB_ProductionProgramActual".Program.St1Insertion[5] )
      { S7_Templates := "SrcType := DInt" } EQ_Contact(in1 := "DB_STATUS_IJCORE".INDEX_MSG_CONFIG, in2 := 1)
      Contact( "IJC_DB".Send_STA[1] )
      S_Coil( "DB_STATUS_IJCORE".CONFIG_MSG[1].START )
   END_RUNG
   RUNG wire#powerrail
      Contact( "DB_ProductionProgramActual".Program.St1Insertion[5] )
      { S7_Templates := "SrcType := DInt" } EQ_Contact(in1 := "DB_STATUS_IJCORE".INDEX_MSG_CONFIG, in2 := 2)
      Contact( "IJC_DB".IJC_Enable )
      wire#w1
      Contact( "IJC_DB".Send_STA[2] )
      wire#w2
      S_Coil( "DB_STATUS_IJCORE".CONFIG_MSG[2].START )
   END_RUNG
   RUNG wire#w1
      { S7_Templates := "SrcType := Int" } GE_Contact(in1 := "IJC_DB".MSG[1].SEQ_STEP, in2 := 60)
      Contact( "READER_MODEL_ACTUAL".SIDE_RH_SCANNER_OK )
   END_RUNG wire#w2
   RUNG wire#powerrail
      Contact( "DB_ProductionProgramActual".Program.St1Insertion[5] )
      { S7_Templates := "SrcType := DInt" } EQ_Contact(in1 := "DB_STATUS_IJCORE".INDEX_MSG_CONFIG, in2 := 3)
      Contact( "READER_MODEL_ACTUAL".PRODUCTO.NUM_TUBE )
      Contact( "IJC_DB".IJC_Enable )
      wire#w3
      Contact( "IJC_DB".Send_STA[3] )
      wire#w4
      S_Coil( "DB_STATUS_IJCORE".CONFIG_MSG[3].START )
   END_RUNG
   RUNG wire#w3
      { S7_Templates := "SrcType := Int" } GE_Contact(in1 := "IJC_DB".MSG[2].SEQ_STEP, in2 := 60)
      Contact( "READER_MODEL_ACTUAL".FRONT_TUBE_SCANNER_OK )
   END_RUNG wire#w4
   RUNG wire#powerrail
      Contact( "DB_ProductionProgramActual".Program.St1Insertion[5] )
      { S7_Templates := "SrcType := DInt" } EQ_Contact(in1 := "DB_STATUS_IJCORE".INDEX_MSG_CONFIG, in2 := 4)
      Contact( "IJC_DB".IJC_Enable )
      wire#w5
      Contact( "IJC_DB".Send_STA[4] )
      wire#w6
      S_Coil( "DB_STATUS_IJCORE".CONFIG_MSG[4].START )
   END_RUNG
   RUNG wire#w5
      { S7_Templates := "SrcType := Int" } GE_Contact(in1 := "IJC_DB".MSG[3].SEQ_STEP, in2 := 60)
      Contact( "READER_MODEL_ACTUAL".REAR_TUBE_SCANNER_OK )
   END_RUNG wire#w6
   // the same network as SCL:
   IF "DB_ProductionProgramActual".Program.St1Insertion[5] AND ("DB_STATUS_IJCORE".INDEX_MSG_CONFIG = 1) AND "IJC_DB".Send_STA[1] THEN
       "DB_STATUS_IJCORE".CONFIG_MSG[1].START := TRUE;
   END_IF;
   IF "DB_ProductionProgramActual".Program.St1Insertion[5] AND ("DB_STATUS_IJCORE".INDEX_MSG_CONFIG = 2) AND "IJC_DB".IJC_Enable AND ("IJC_DB".Send_STA[2] OR (("IJC_DB".MSG[1].SEQ_STEP >= 60) AND "READER_MODEL_ACTUAL".SIDE_RH_SCANNER_OK)) THEN
       "DB_STATUS_IJCORE".CONFIG_MSG[2].START := TRUE;
   END_IF;
   IF "DB_ProductionProgramActual".Program.St1Insertion[5] AND ("DB_STATUS_IJCORE".INDEX_MSG_CONFIG = 3) AND "READER_MODEL_ACTUAL".PRODUCTO.NUM_TUBE AND "IJC_DB".IJC_Enable AND ("IJC_DB".Send_STA[3] OR (("IJC_DB".MSG[2].SEQ_STEP >= 60) AND "READER_MODEL_ACTUAL".FRONT_TUBE_SCANNER_OK)) THEN
       "DB_STATUS_IJCORE".CONFIG_MSG[3].START := TRUE;
   END_IF;
   IF "DB_ProductionProgramActual".Program.St1Insertion[5] AND ("DB_STATUS_IJCORE".INDEX_MSG_CONFIG = 4) AND "IJC_DB".IJC_Enable AND ("IJC_DB".Send_STA[4] OR (("IJC_DB".MSG[3].SEQ_STEP >= 60) AND "READER_MODEL_ACTUAL".REAR_TUBE_SCANNER_OK)) THEN
       "DB_STATUS_IJCORE".CONFIG_MSG[4].START := TRUE;
   END_IF;
END_REGION

REGION Network 12: SEND TRC SCAN LABEL
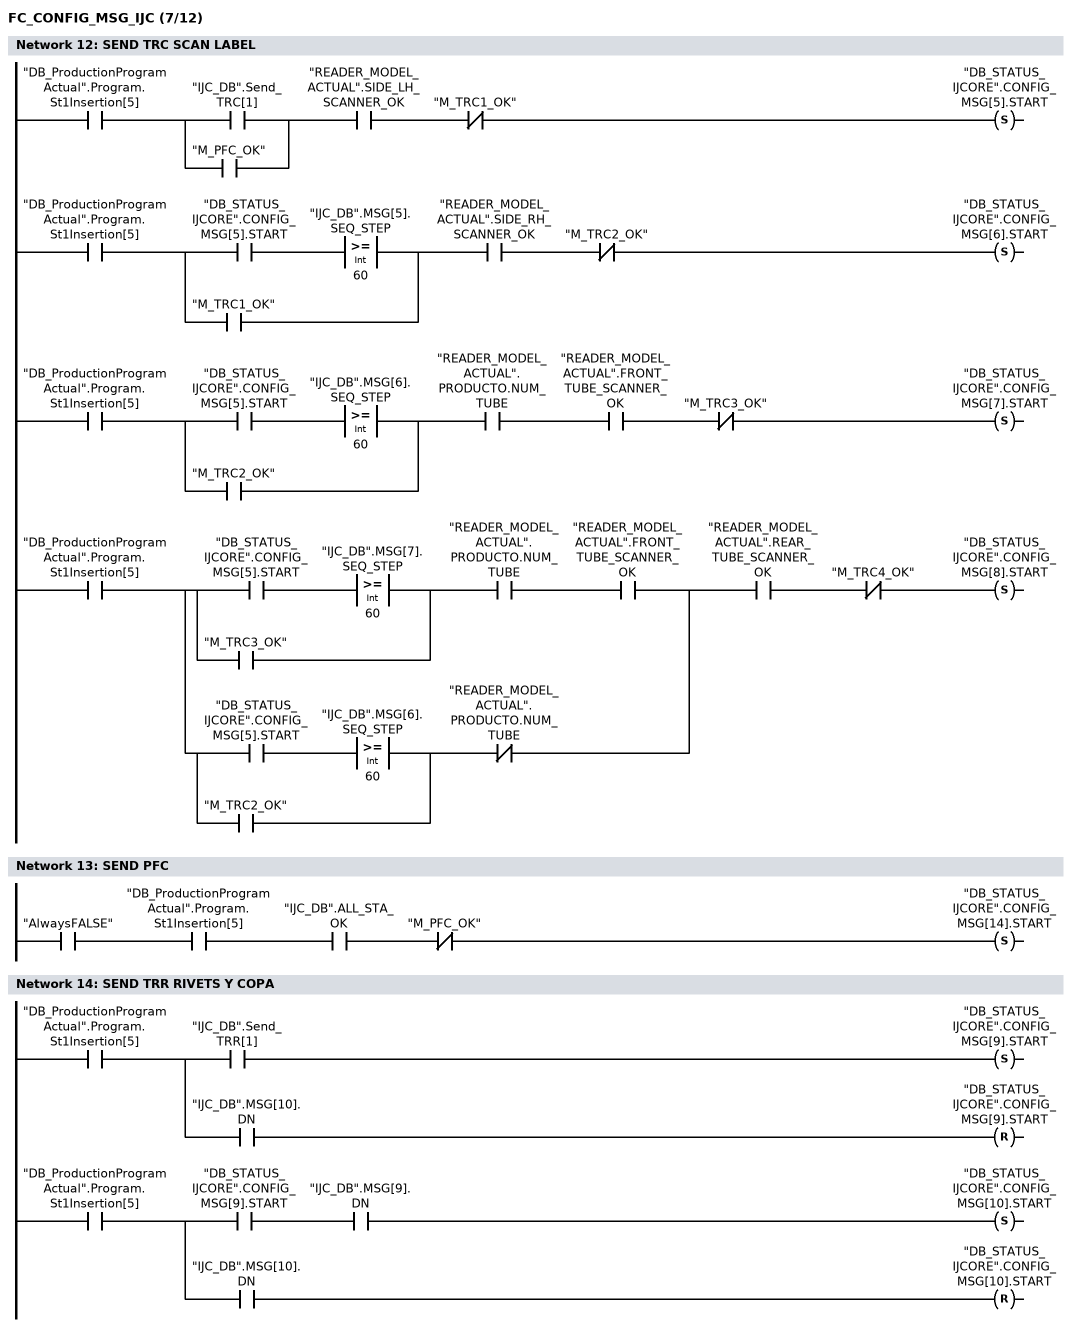
   RUNG wire#powerrail
      Contact( "DB_ProductionProgramActual".Program.St1Insertion[5] )
      wire#w1
      Contact( "IJC_DB".Send_TRC[1] )
      wire#w2
      Contact( "READER_MODEL_ACTUAL".SIDE_LH_SCANNER_OK )
      I_Contact( "M_TRC1_OK" )
      S_Coil( "DB_STATUS_IJCORE".CONFIG_MSG[5].START )
   END_RUNG
   RUNG wire#w1
      Contact( "M_PFC_OK" )
   END_RUNG wire#w2
   RUNG wire#powerrail
      Contact( "DB_ProductionProgramActual".Program.St1Insertion[5] )
      wire#w3
      Contact( "DB_STATUS_IJCORE".CONFIG_MSG[5].START )
      { S7_Templates := "SrcType := Int" } GE_Contact(in1 := "IJC_DB".MSG[5].SEQ_STEP, in2 := 60)
      wire#w4
      Contact( "READER_MODEL_ACTUAL".SIDE_RH_SCANNER_OK )
      I_Contact( "M_TRC2_OK" )
      S_Coil( "DB_STATUS_IJCORE".CONFIG_MSG[6].START )
   END_RUNG
   RUNG wire#w3
      Contact( "M_TRC1_OK" )
   END_RUNG wire#w4
   RUNG wire#powerrail
      Contact( "DB_ProductionProgramActual".Program.St1Insertion[5] )
      wire#w5
      Contact( "DB_STATUS_IJCORE".CONFIG_MSG[5].START )
      { S7_Templates := "SrcType := Int" } GE_Contact(in1 := "IJC_DB".MSG[6].SEQ_STEP, in2 := 60)
      wire#w6
      Contact( "READER_MODEL_ACTUAL".PRODUCTO.NUM_TUBE )
      Contact( "READER_MODEL_ACTUAL".FRONT_TUBE_SCANNER_OK )
      I_Contact( "M_TRC3_OK" )
      S_Coil( "DB_STATUS_IJCORE".CONFIG_MSG[7].START )
   END_RUNG
   RUNG wire#w5
      Contact( "M_TRC2_OK" )
   END_RUNG wire#w6
   RUNG wire#powerrail
      Contact( "DB_ProductionProgramActual".Program.St1Insertion[5] )
      wire#w7
      Contact( "DB_STATUS_IJCORE".CONFIG_MSG[5].START )
      { S7_Templates := "SrcType := Int" } GE_Contact(in1 := "IJC_DB".MSG[7].SEQ_STEP, in2 := 60)
      wire#w8
      Contact( "READER_MODEL_ACTUAL".PRODUCTO.NUM_TUBE )
      Contact( "READER_MODEL_ACTUAL".FRONT_TUBE_SCANNER_OK )
      wire#w9
      Contact( "READER_MODEL_ACTUAL".REAR_TUBE_SCANNER_OK )
      I_Contact( "M_TRC4_OK" )
      S_Coil( "DB_STATUS_IJCORE".CONFIG_MSG[8].START )
   END_RUNG
   RUNG wire#w7
      Contact( "M_TRC3_OK" )
   END_RUNG wire#w8
   RUNG wire#w7
      Contact( "DB_STATUS_IJCORE".CONFIG_MSG[5].START )
      { S7_Templates := "SrcType := Int" } GE_Contact(in1 := "IJC_DB".MSG[6].SEQ_STEP, in2 := 60)
      wire#w10
      I_Contact( "READER_MODEL_ACTUAL".PRODUCTO.NUM_TUBE )
   END_RUNG wire#w9
   RUNG wire#w7
      Contact( "M_TRC2_OK" )
   END_RUNG wire#w10
   // the same network as SCL:
   IF "DB_ProductionProgramActual".Program.St1Insertion[5] AND ("IJC_DB".Send_TRC[1] OR "M_PFC_OK") AND "READER_MODEL_ACTUAL".SIDE_LH_SCANNER_OK AND NOT "M_TRC1_OK" THEN
       "DB_STATUS_IJCORE".CONFIG_MSG[5].START := TRUE;
   END_IF;
   IF "DB_ProductionProgramActual".Program.St1Insertion[5] AND (("DB_STATUS_IJCORE".CONFIG_MSG[5].START AND ("IJC_DB".MSG[5].SEQ_STEP >= 60)) OR "M_TRC1_OK") AND "READER_MODEL_ACTUAL".SIDE_RH_SCANNER_OK AND NOT "M_TRC2_OK" THEN
       "DB_STATUS_IJCORE".CONFIG_MSG[6].START := TRUE;
   END_IF;
   IF "DB_ProductionProgramActual".Program.St1Insertion[5] AND (("DB_STATUS_IJCORE".CONFIG_MSG[5].START AND ("IJC_DB".MSG[6].SEQ_STEP >= 60)) OR "M_TRC2_OK") AND "READER_MODEL_ACTUAL".PRODUCTO.NUM_TUBE AND "READER_MODEL_ACTUAL".FRONT_TUBE_SCANNER_OK AND NOT "M_TRC3_OK" THEN
       "DB_STATUS_IJCORE".CONFIG_MSG[7].START := TRUE;
   END_IF;
   IF "DB_ProductionProgramActual".Program.St1Insertion[5] AND (((("DB_STATUS_IJCORE".CONFIG_MSG[5].START AND ("IJC_DB".MSG[7].SEQ_STEP >= 60)) OR "M_TRC3_OK") AND "READER_MODEL_ACTUAL".PRODUCTO.NUM_TUBE AND "READER_MODEL_ACTUAL".FRONT_TUBE_SCANNER_OK) OR ((("DB_STATUS_IJCORE".CONFIG_MSG[5].START AND ("IJC_DB".MSG[6].SEQ_STEP >= 60)) OR "M_TRC2_OK") AND NOT "READER_MODEL_ACTUAL".PRODUCTO.NUM_TUBE)) AND "READER_MODEL_ACTUAL".REAR_TUBE_SCANNER_OK AND NOT "M_TRC4_OK" THEN
       "DB_STATUS_IJCORE".CONFIG_MSG[8].START := TRUE;
   END_IF;
END_REGION

REGION Network 13: SEND PFC
   RUNG wire#powerrail
      Contact( "AlwaysFALSE" )
      Contact( "DB_ProductionProgramActual".Program.St1Insertion[5] )
      Contact( "IJC_DB".ALL_STA_OK )
      I_Contact( "M_PFC_OK" )
      S_Coil( "DB_STATUS_IJCORE".CONFIG_MSG[14].START )
   END_RUNG
   // the same network as SCL:
   IF "AlwaysFALSE" AND "DB_ProductionProgramActual".Program.St1Insertion[5] AND "IJC_DB".ALL_STA_OK AND NOT "M_PFC_OK" THEN
       "DB_STATUS_IJCORE".CONFIG_MSG[14].START := TRUE;
   END_IF;
END_REGION

REGION Network 14: SEND TRR RIVETS Y COPA
   RUNG wire#powerrail
      Contact( "DB_ProductionProgramActual".Program.St1Insertion[5] )
      wire#w1
      Contact( "IJC_DB".Send_TRR[1] )
      S_Coil( "DB_STATUS_IJCORE".CONFIG_MSG[9].START )
   END_RUNG
   RUNG wire#w1
      Contact( "IJC_DB".MSG[10].DN )
      R_Coil( "DB_STATUS_IJCORE".CONFIG_MSG[9].START )
   END_RUNG
   RUNG wire#powerrail
      Contact( "DB_ProductionProgramActual".Program.St1Insertion[5] )
      wire#w2
      Contact( "DB_STATUS_IJCORE".CONFIG_MSG[9].START )
      Contact( "IJC_DB".MSG[9].DN )
      S_Coil( "DB_STATUS_IJCORE".CONFIG_MSG[10].START )
   END_RUNG
   RUNG wire#w2
      Contact( "IJC_DB".MSG[10].DN )
      R_Coil( "DB_STATUS_IJCORE".CONFIG_MSG[10].START )
   END_RUNG
   // the same network as SCL:
   IF "DB_ProductionProgramActual".Program.St1Insertion[5] AND "IJC_DB".Send_TRR[1] THEN
       "DB_STATUS_IJCORE".CONFIG_MSG[9].START := TRUE;
   END_IF;
   IF "DB_ProductionProgramActual".Program.St1Insertion[5] AND "IJC_DB".MSG[10].DN THEN
       "DB_STATUS_IJCORE".CONFIG_MSG[9].START := FALSE;
   END_IF;
   IF "DB_ProductionProgramActual".Program.St1Insertion[5] AND "DB_STATUS_IJCORE".CONFIG_MSG[9].START AND "IJC_DB".MSG[9].DN THEN
       "DB_STATUS_IJCORE".CONFIG_MSG[10].START := TRUE;
   END_IF;
   IF "DB_ProductionProgramActual".Program.St1Insertion[5] AND "IJC_DB".MSG[10].DN THEN
       "DB_STATUS_IJCORE".CONFIG_MSG[10].START := FALSE;
   END_IF;
END_REGION

REGION Network 15: SEND CNF
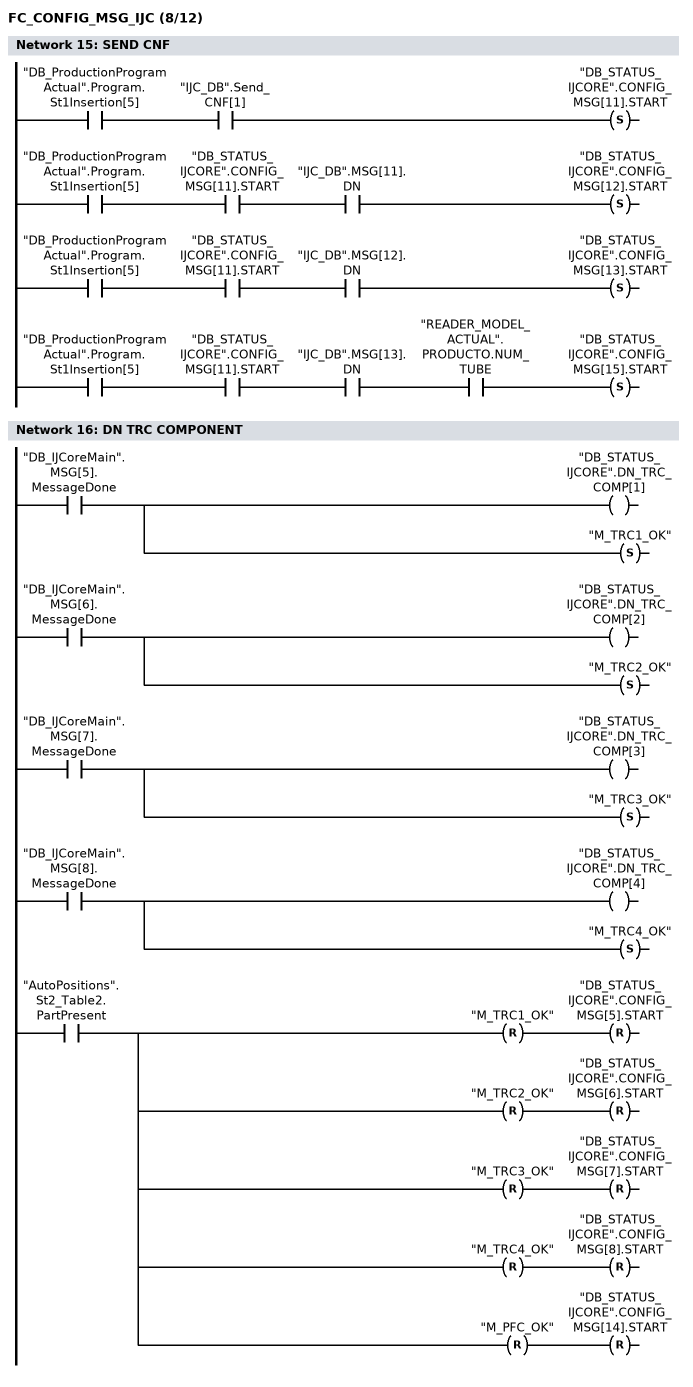
   RUNG wire#powerrail
      Contact( "DB_ProductionProgramActual".Program.St1Insertion[5] )
      Contact( "IJC_DB".Send_CNF[1] )
      S_Coil( "DB_STATUS_IJCORE".CONFIG_MSG[11].START )
   END_RUNG
   RUNG wire#powerrail
      Contact( "DB_ProductionProgramActual".Program.St1Insertion[5] )
      Contact( "DB_STATUS_IJCORE".CONFIG_MSG[11].START )
      Contact( "IJC_DB".MSG[11].DN )
      S_Coil( "DB_STATUS_IJCORE".CONFIG_MSG[12].START )
   END_RUNG
   RUNG wire#powerrail
      Contact( "DB_ProductionProgramActual".Program.St1Insertion[5] )
      Contact( "DB_STATUS_IJCORE".CONFIG_MSG[11].START )
      Contact( "IJC_DB".MSG[12].DN )
      S_Coil( "DB_STATUS_IJCORE".CONFIG_MSG[13].START )
   END_RUNG
   RUNG wire#powerrail
      Contact( "DB_ProductionProgramActual".Program.St1Insertion[5] )
      Contact( "DB_STATUS_IJCORE".CONFIG_MSG[11].START )
      Contact( "IJC_DB".MSG[13].DN )
      Contact( "READER_MODEL_ACTUAL".PRODUCTO.NUM_TUBE )
      S_Coil( "DB_STATUS_IJCORE".CONFIG_MSG[15].START )
   END_RUNG
   // the same network as SCL:
   IF "DB_ProductionProgramActual".Program.St1Insertion[5] AND "IJC_DB".Send_CNF[1] THEN
       "DB_STATUS_IJCORE".CONFIG_MSG[11].START := TRUE;
   END_IF;
   IF "DB_ProductionProgramActual".Program.St1Insertion[5] AND "DB_STATUS_IJCORE".CONFIG_MSG[11].START AND "IJC_DB".MSG[11].DN THEN
       "DB_STATUS_IJCORE".CONFIG_MSG[12].START := TRUE;
   END_IF;
   IF "DB_ProductionProgramActual".Program.St1Insertion[5] AND "DB_STATUS_IJCORE".CONFIG_MSG[11].START AND "IJC_DB".MSG[12].DN THEN
       "DB_STATUS_IJCORE".CONFIG_MSG[13].START := TRUE;
   END_IF;
   IF "DB_ProductionProgramActual".Program.St1Insertion[5] AND "DB_STATUS_IJCORE".CONFIG_MSG[11].START AND "IJC_DB".MSG[13].DN AND "READER_MODEL_ACTUAL".PRODUCTO.NUM_TUBE THEN
       "DB_STATUS_IJCORE".CONFIG_MSG[15].START := TRUE;
   END_IF;
END_REGION

REGION Network 16: DN TRC COMPONENT
   RUNG wire#powerrail
      Contact( "DB_IJCoreMain".MSG[5].MessageDone )
      wire#w1
      Coil( "DB_STATUS_IJCORE".DN_TRC_COMP[1] )
   END_RUNG
   RUNG wire#w1
      S_Coil( "M_TRC1_OK" )
   END_RUNG
   RUNG wire#powerrail
      Contact( "DB_IJCoreMain".MSG[6].MessageDone )
      wire#w2
      Coil( "DB_STATUS_IJCORE".DN_TRC_COMP[2] )
   END_RUNG
   RUNG wire#w2
      S_Coil( "M_TRC2_OK" )
   END_RUNG
   RUNG wire#powerrail
      Contact( "DB_IJCoreMain".MSG[7].MessageDone )
      wire#w3
      Coil( "DB_STATUS_IJCORE".DN_TRC_COMP[3] )
   END_RUNG
   RUNG wire#w3
      S_Coil( "M_TRC3_OK" )
   END_RUNG
   RUNG wire#powerrail
      Contact( "DB_IJCoreMain".MSG[8].MessageDone )
      wire#w4
      Coil( "DB_STATUS_IJCORE".DN_TRC_COMP[4] )
   END_RUNG
   RUNG wire#w4
      S_Coil( "M_TRC4_OK" )
   END_RUNG
   RUNG wire#powerrail
      Contact( "AutoPositions".St2_Table2.PartPresent )
      wire#w5
      R_Coil( "M_TRC1_OK" )
      R_Coil( "DB_STATUS_IJCORE".CONFIG_MSG[5].START )
   END_RUNG
   RUNG wire#w5
      R_Coil( "M_TRC2_OK" )
      R_Coil( "DB_STATUS_IJCORE".CONFIG_MSG[6].START )
   END_RUNG
   RUNG wire#w5
      R_Coil( "M_TRC3_OK" )
      R_Coil( "DB_STATUS_IJCORE".CONFIG_MSG[7].START )
   END_RUNG
   RUNG wire#w5
      R_Coil( "M_TRC4_OK" )
      R_Coil( "DB_STATUS_IJCORE".CONFIG_MSG[8].START )
   END_RUNG
   RUNG wire#w5
      R_Coil( "M_PFC_OK" )
      R_Coil( "DB_STATUS_IJCORE".CONFIG_MSG[14].START )
   END_RUNG
   // the same network as SCL:
   "DB_STATUS_IJCORE".DN_TRC_COMP[1] := "DB_IJCoreMain".MSG[5].MessageDone;
   IF "DB_IJCoreMain".MSG[5].MessageDone THEN "M_TRC1_OK" := TRUE; END_IF;
   "DB_STATUS_IJCORE".DN_TRC_COMP[2] := "DB_IJCoreMain".MSG[6].MessageDone;
   IF "DB_IJCoreMain".MSG[6].MessageDone THEN "M_TRC2_OK" := TRUE; END_IF;
   "DB_STATUS_IJCORE".DN_TRC_COMP[3] := "DB_IJCoreMain".MSG[7].MessageDone;
   IF "DB_IJCoreMain".MSG[7].MessageDone THEN "M_TRC3_OK" := TRUE; END_IF;
   "DB_STATUS_IJCORE".DN_TRC_COMP[4] := "DB_IJCoreMain".MSG[8].MessageDone;
   IF "DB_IJCoreMain".MSG[8].MessageDone THEN "M_TRC4_OK" := TRUE; END_IF;
   IF "AutoPositions".St2_Table2.PartPresent THEN
       "M_TRC1_OK" := FALSE;
       "DB_STATUS_IJCORE".CONFIG_MSG[5].START := FALSE;
       "M_TRC2_OK" := FALSE;
       "DB_STATUS_IJCORE".CONFIG_MSG[6].START := FALSE;
       "M_TRC3_OK" := FALSE;
       "DB_STATUS_IJCORE".CONFIG_MSG[7].START := FALSE;
       "M_TRC4_OK" := FALSE;
       "DB_STATUS_IJCORE".CONFIG_MSG[8].START := FALSE;
       "M_PFC_OK" := FALSE;
       "DB_STATUS_IJCORE".CONFIG_MSG[14].START := FALSE;
   END_IF;
END_REGION

REGION Network 17: DN STA
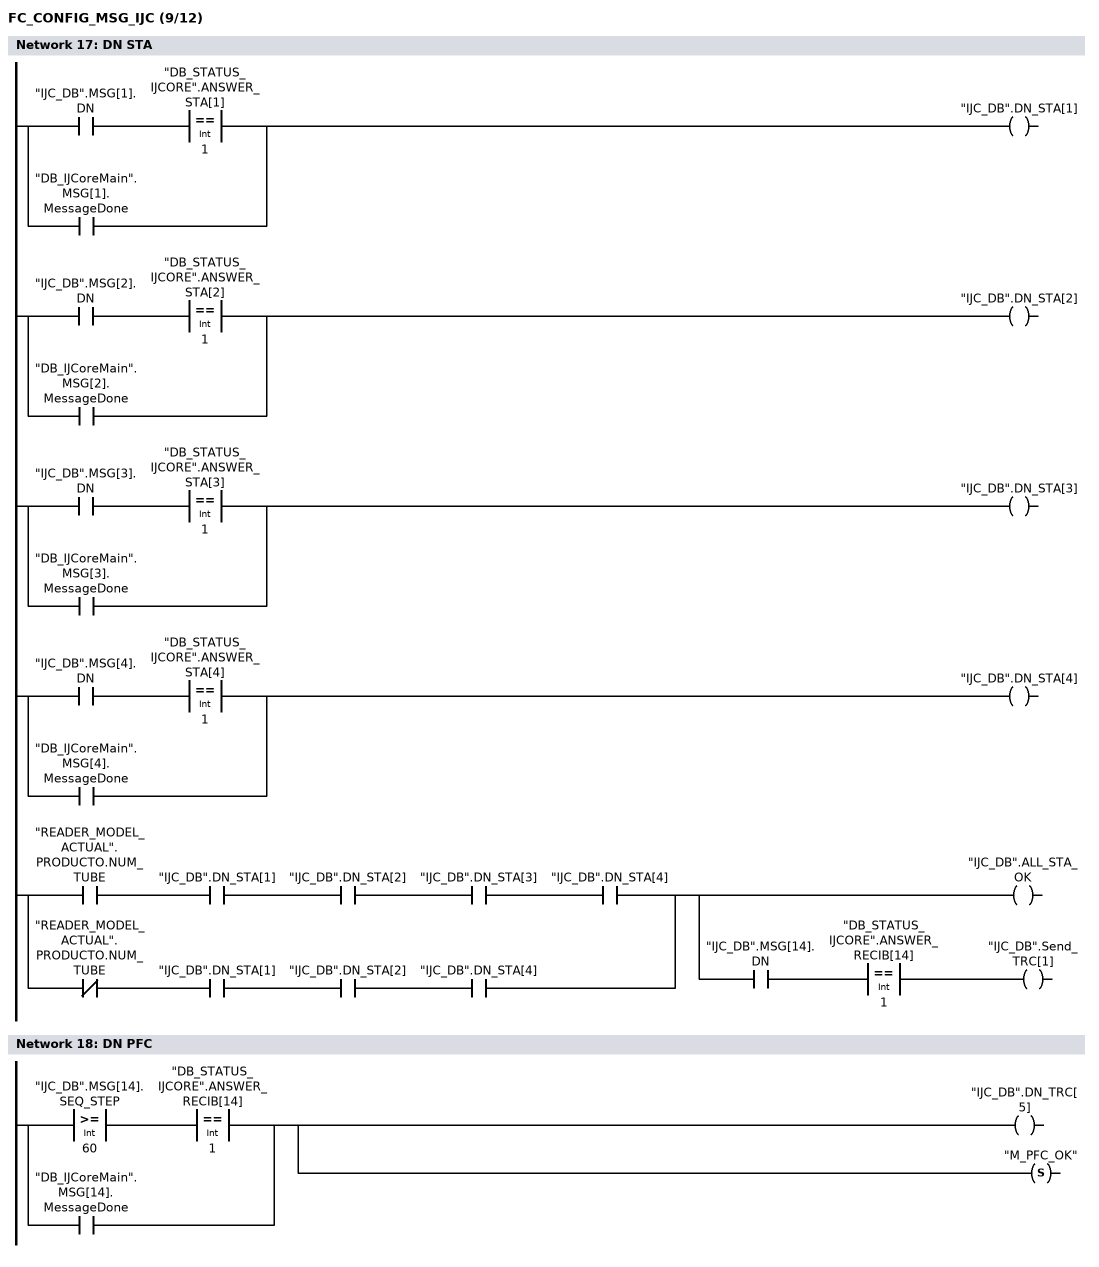
   RUNG wire#powerrail
      Contact( "IJC_DB".MSG[1].DN )
      { S7_Templates := "SrcType := Int" } EQ_Contact(in1 := "DB_STATUS_IJCORE".ANSWER_STA[1], in2 := 1)
      wire#w1
      Coil( "IJC_DB".DN_STA[1] )
   END_RUNG
   RUNG wire#powerrail
      Contact( "DB_IJCoreMain".MSG[1].MessageDone )
   END_RUNG wire#w1
   RUNG wire#powerrail
      Contact( "IJC_DB".MSG[2].DN )
      { S7_Templates := "SrcType := Int" } EQ_Contact(in1 := "DB_STATUS_IJCORE".ANSWER_STA[2], in2 := 1)
      wire#w2
      Coil( "IJC_DB".DN_STA[2] )
   END_RUNG
   RUNG wire#powerrail
      Contact( "DB_IJCoreMain".MSG[2].MessageDone )
   END_RUNG wire#w2
   RUNG wire#powerrail
      Contact( "IJC_DB".MSG[3].DN )
      { S7_Templates := "SrcType := Int" } EQ_Contact(in1 := "DB_STATUS_IJCORE".ANSWER_STA[3], in2 := 1)
      wire#w3
      Coil( "IJC_DB".DN_STA[3] )
   END_RUNG
   RUNG wire#powerrail
      Contact( "DB_IJCoreMain".MSG[3].MessageDone )
   END_RUNG wire#w3
   RUNG wire#powerrail
      Contact( "IJC_DB".MSG[4].DN )
      { S7_Templates := "SrcType := Int" } EQ_Contact(in1 := "DB_STATUS_IJCORE".ANSWER_STA[4], in2 := 1)
      wire#w4
      Coil( "IJC_DB".DN_STA[4] )
   END_RUNG
   RUNG wire#powerrail
      Contact( "DB_IJCoreMain".MSG[4].MessageDone )
   END_RUNG wire#w4
   RUNG wire#powerrail
      Contact( "READER_MODEL_ACTUAL".PRODUCTO.NUM_TUBE )
      Contact( "IJC_DB".DN_STA[1] )
      Contact( "IJC_DB".DN_STA[2] )
      Contact( "IJC_DB".DN_STA[3] )
      Contact( "IJC_DB".DN_STA[4] )
      wire#w5
      Coil( "IJC_DB".ALL_STA_OK )
   END_RUNG
   RUNG wire#powerrail
      I_Contact( "READER_MODEL_ACTUAL".PRODUCTO.NUM_TUBE )
      Contact( "IJC_DB".DN_STA[1] )
      Contact( "IJC_DB".DN_STA[2] )
      Contact( "IJC_DB".DN_STA[4] )
   END_RUNG wire#w5
   RUNG wire#w5
      Contact( "IJC_DB".MSG[14].DN )
      { S7_Templates := "SrcType := Int" } EQ_Contact(in1 := "DB_STATUS_IJCORE".ANSWER_RECIB[14], in2 := 1)
      Coil( "IJC_DB".Send_TRC[1] )
   END_RUNG
   // the same network as SCL:
   "IJC_DB".DN_STA[1] := ("IJC_DB".MSG[1].DN AND ("DB_STATUS_IJCORE".ANSWER_STA[1] = 1)) OR "DB_IJCoreMain".MSG[1].MessageDone;
   "IJC_DB".DN_STA[2] := ("IJC_DB".MSG[2].DN AND ("DB_STATUS_IJCORE".ANSWER_STA[2] = 1)) OR "DB_IJCoreMain".MSG[2].MessageDone;
   "IJC_DB".DN_STA[3] := ("IJC_DB".MSG[3].DN AND ("DB_STATUS_IJCORE".ANSWER_STA[3] = 1)) OR "DB_IJCoreMain".MSG[3].MessageDone;
   "IJC_DB".DN_STA[4] := ("IJC_DB".MSG[4].DN AND ("DB_STATUS_IJCORE".ANSWER_STA[4] = 1)) OR "DB_IJCoreMain".MSG[4].MessageDone;
   "IJC_DB".ALL_STA_OK := ("READER_MODEL_ACTUAL".PRODUCTO.NUM_TUBE AND "IJC_DB".DN_STA[1] AND "IJC_DB".DN_STA[2] AND "IJC_DB".DN_STA[3] AND "IJC_DB".DN_STA[4]) OR (NOT "READER_MODEL_ACTUAL".PRODUCTO.NUM_TUBE AND "IJC_DB".DN_STA[1] AND "IJC_DB".DN_STA[2] AND "IJC_DB".DN_STA[4]);
   "IJC_DB".Send_TRC[1] := "IJC_DB".ALL_STA_OK AND "IJC_DB".MSG[14].DN AND ("DB_STATUS_IJCORE".ANSWER_RECIB[14] = 1);
END_REGION

REGION Network 18: DN PFC
   RUNG wire#powerrail
      { S7_Templates := "SrcType := Int" } GE_Contact(in1 := "IJC_DB".MSG[14].SEQ_STEP, in2 := 60)
      { S7_Templates := "SrcType := Int" } EQ_Contact(in1 := "DB_STATUS_IJCORE".ANSWER_RECIB[14], in2 := 1)
      wire#w1
      Coil( "IJC_DB".DN_TRC[5] )
   END_RUNG
   RUNG wire#powerrail
      Contact( "DB_IJCoreMain".MSG[14].MessageDone )
   END_RUNG wire#w1
   RUNG wire#w1
      S_Coil( "M_PFC_OK" )
   END_RUNG
   // the same network as SCL:
   "IJC_DB".DN_TRC[5] := (("IJC_DB".MSG[14].SEQ_STEP >= 60) AND ("DB_STATUS_IJCORE".ANSWER_RECIB[14] = 1)) OR "DB_IJCoreMain".MSG[14].MessageDone;
   IF (("IJC_DB".MSG[14].SEQ_STEP >= 60) AND ("DB_STATUS_IJCORE".ANSWER_RECIB[14] = 1)) OR "DB_IJCoreMain".MSG[14].MessageDone THEN
       "M_PFC_OK" := TRUE;
   END_IF;
END_REGION

REGION Network 19: DN TRR
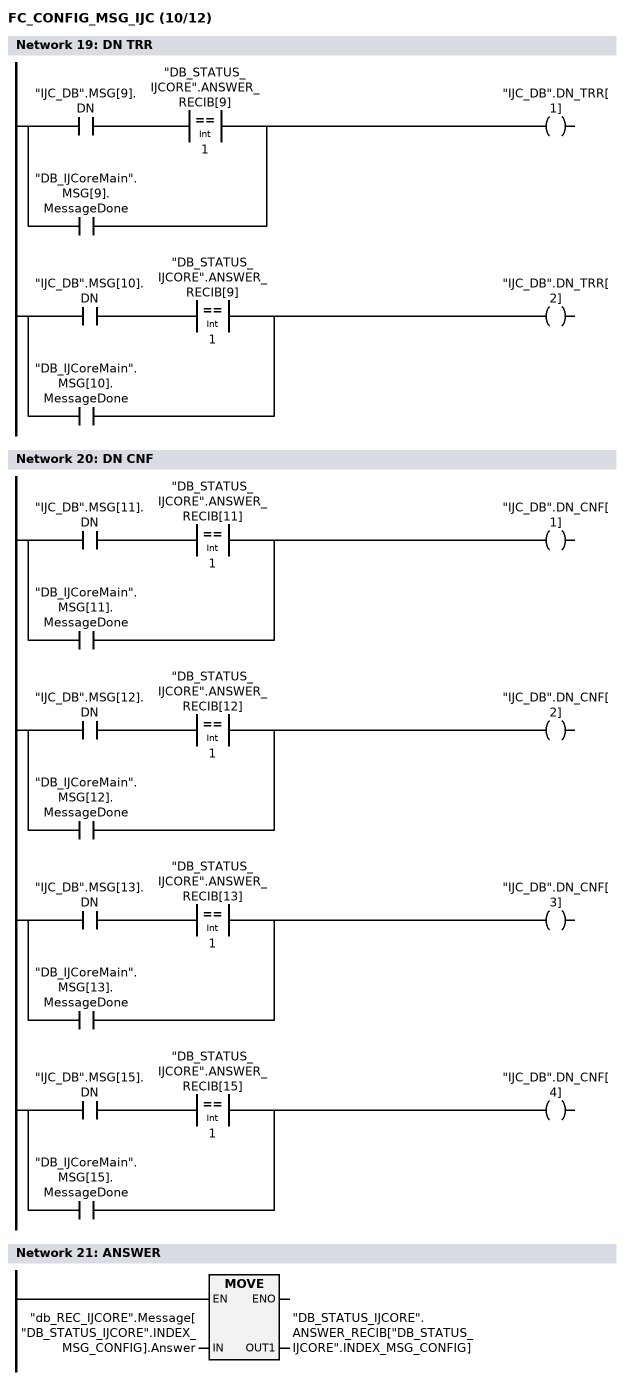
   RUNG wire#powerrail
      Contact( "IJC_DB".MSG[9].DN )
      { S7_Templates := "SrcType := Int" } EQ_Contact(in1 := "DB_STATUS_IJCORE".ANSWER_RECIB[9], in2 := 1)
      wire#w1
      Coil( "IJC_DB".DN_TRR[1] )
   END_RUNG
   RUNG wire#powerrail
      Contact( "DB_IJCoreMain".MSG[9].MessageDone )
   END_RUNG wire#w1
   RUNG wire#powerrail
      Contact( "IJC_DB".MSG[10].DN )
      { S7_Templates := "SrcType := Int" } EQ_Contact(in1 := "DB_STATUS_IJCORE".ANSWER_RECIB[9], in2 := 1)
      wire#w2
      Coil( "IJC_DB".DN_TRR[2] )
   END_RUNG
   RUNG wire#powerrail
      Contact( "DB_IJCoreMain".MSG[10].MessageDone )
   END_RUNG wire#w2
   // the same network as SCL:
   "IJC_DB".DN_TRR[1] := ("IJC_DB".MSG[9].DN AND ("DB_STATUS_IJCORE".ANSWER_RECIB[9] = 1)) OR "DB_IJCoreMain".MSG[9].MessageDone;
   "IJC_DB".DN_TRR[2] := ("IJC_DB".MSG[10].DN AND ("DB_STATUS_IJCORE".ANSWER_RECIB[9] = 1)) OR "DB_IJCoreMain".MSG[10].MessageDone;
END_REGION

REGION Network 20: DN CNF
   RUNG wire#powerrail
      Contact( "IJC_DB".MSG[11].DN )
      { S7_Templates := "SrcType := Int" } EQ_Contact(in1 := "DB_STATUS_IJCORE".ANSWER_RECIB[11], in2 := 1)
      wire#w1
      Coil( "IJC_DB".DN_CNF[1] )
   END_RUNG
   RUNG wire#powerrail
      Contact( "DB_IJCoreMain".MSG[11].MessageDone )
   END_RUNG wire#w1
   RUNG wire#powerrail
      Contact( "IJC_DB".MSG[12].DN )
      { S7_Templates := "SrcType := Int" } EQ_Contact(in1 := "DB_STATUS_IJCORE".ANSWER_RECIB[12], in2 := 1)
      wire#w2
      Coil( "IJC_DB".DN_CNF[2] )
   END_RUNG
   RUNG wire#powerrail
      Contact( "DB_IJCoreMain".MSG[12].MessageDone )
   END_RUNG wire#w2
   RUNG wire#powerrail
      Contact( "IJC_DB".MSG[13].DN )
      { S7_Templates := "SrcType := Int" } EQ_Contact(in1 := "DB_STATUS_IJCORE".ANSWER_RECIB[13], in2 := 1)
      wire#w3
      Coil( "IJC_DB".DN_CNF[3] )
   END_RUNG
   RUNG wire#powerrail
      Contact( "DB_IJCoreMain".MSG[13].MessageDone )
   END_RUNG wire#w3
   RUNG wire#powerrail
      Contact( "IJC_DB".MSG[15].DN )
      { S7_Templates := "SrcType := Int" } EQ_Contact(in1 := "DB_STATUS_IJCORE".ANSWER_RECIB[15], in2 := 1)
      wire#w4
      Coil( "IJC_DB".DN_CNF[4] )
   END_RUNG
   RUNG wire#powerrail
      Contact( "DB_IJCoreMain".MSG[15].MessageDone )
   END_RUNG wire#w4
   // the same network as SCL:
   "IJC_DB".DN_CNF[1] := ("IJC_DB".MSG[11].DN AND ("DB_STATUS_IJCORE".ANSWER_RECIB[11] = 1)) OR "DB_IJCoreMain".MSG[11].MessageDone;
   "IJC_DB".DN_CNF[2] := ("IJC_DB".MSG[12].DN AND ("DB_STATUS_IJCORE".ANSWER_RECIB[12] = 1)) OR "DB_IJCoreMain".MSG[12].MessageDone;
   "IJC_DB".DN_CNF[3] := ("IJC_DB".MSG[13].DN AND ("DB_STATUS_IJCORE".ANSWER_RECIB[13] = 1)) OR "DB_IJCoreMain".MSG[13].MessageDone;
   "IJC_DB".DN_CNF[4] := ("IJC_DB".MSG[15].DN AND ("DB_STATUS_IJCORE".ANSWER_RECIB[15] = 1)) OR "DB_IJCoreMain".MSG[15].MessageDone;
END_REGION

REGION Network 21: ANSWER
   RUNG wire#powerrail
      Move(in := "db_REC_IJCORE".Message["DB_STATUS_IJCORE".INDEX_MSG_CONFIG].Answer, out1 => "DB_STATUS_IJCORE".ANSWER_RECIB["DB_STATUS_IJCORE".INDEX_MSG_CONFIG])
   END_RUNG
   // the same network as SCL:
   "DB_STATUS_IJCORE".ANSWER_RECIB["DB_STATUS_IJCORE".INDEX_MSG_CONFIG] := "db_REC_IJCORE".Message["DB_STATUS_IJCORE".INDEX_MSG_CONFIG].Answer;
END_REGION

REGION Network 22: ANSWER NFP
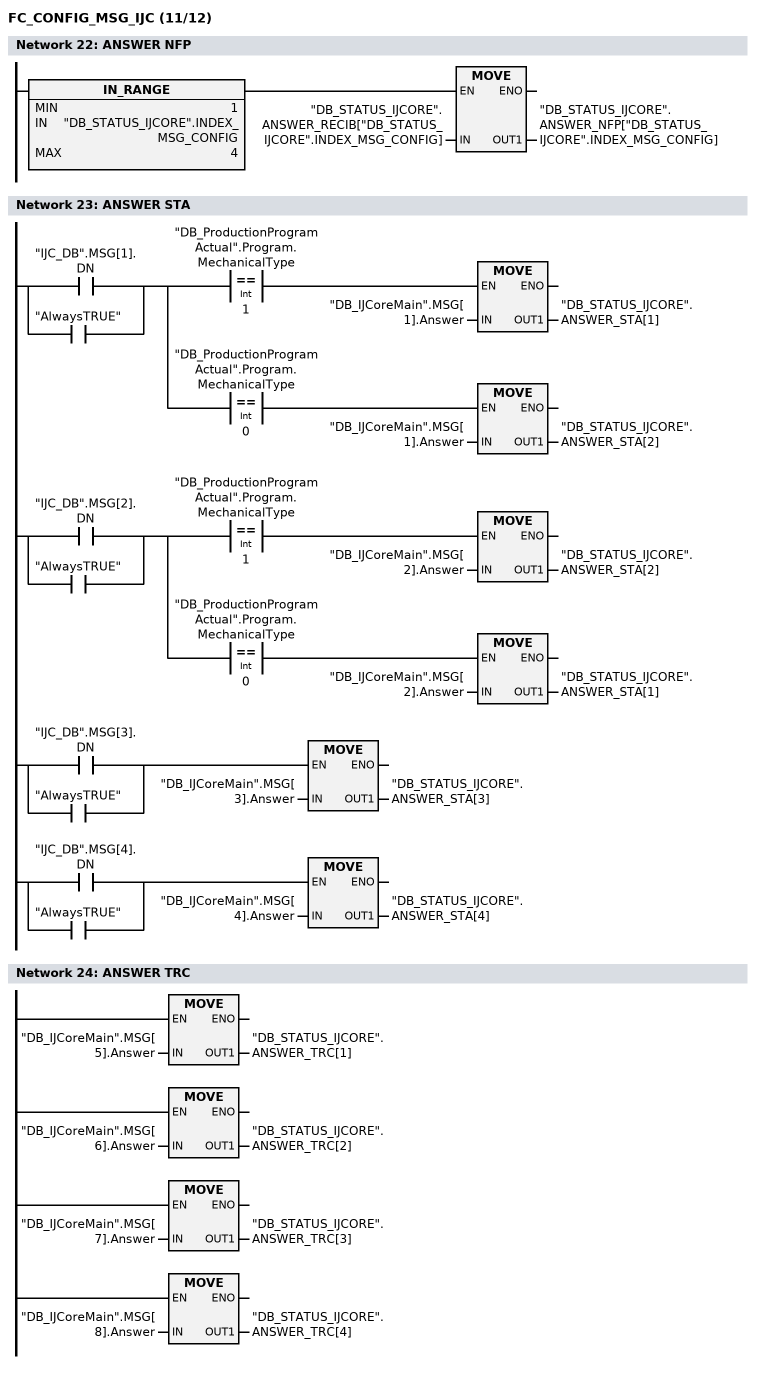
   RUNG wire#powerrail
      { S7_Templates := "SrcType := DInt" } InRange(min := 1, in := "DB_STATUS_IJCORE".INDEX_MSG_CONFIG, max := 4)
      Move(in := "DB_STATUS_IJCORE".ANSWER_RECIB["DB_STATUS_IJCORE".INDEX_MSG_CONFIG], out1 => "DB_STATUS_IJCORE".ANSWER_NFP["DB_STATUS_IJCORE".INDEX_MSG_CONFIG])
   END_RUNG
   // the same network as SCL:
   IF (1 <= "DB_STATUS_IJCORE".INDEX_MSG_CONFIG) AND ("DB_STATUS_IJCORE".INDEX_MSG_CONFIG <= 4) THEN
       "DB_STATUS_IJCORE".ANSWER_NFP["DB_STATUS_IJCORE".INDEX_MSG_CONFIG] := "DB_STATUS_IJCORE".ANSWER_RECIB["DB_STATUS_IJCORE".INDEX_MSG_CONFIG];
   END_IF;
END_REGION

REGION Network 23: ANSWER STA
   RUNG wire#powerrail
      Contact( "IJC_DB".MSG[1].DN )
      wire#w1
      { S7_Templates := "SrcType := Int" } EQ_Contact(in1 := "DB_ProductionProgramActual".Program.MechanicalType, in2 := 1)
      Move(in := "DB_IJCoreMain".MSG[1].Answer, out1 => "DB_STATUS_IJCORE".ANSWER_STA[1])
   END_RUNG
   RUNG wire#powerrail
      Contact( "AlwaysTRUE" )
   END_RUNG wire#w1
   RUNG wire#w1
      { S7_Templates := "SrcType := Int" } EQ_Contact(in1 := "DB_ProductionProgramActual".Program.MechanicalType, in2 := 0)
      Move(in := "DB_IJCoreMain".MSG[1].Answer, out1 => "DB_STATUS_IJCORE".ANSWER_STA[2])
   END_RUNG
   RUNG wire#powerrail
      Contact( "IJC_DB".MSG[2].DN )
      wire#w2
      { S7_Templates := "SrcType := Int" } EQ_Contact(in1 := "DB_ProductionProgramActual".Program.MechanicalType, in2 := 1)
      Move(in := "DB_IJCoreMain".MSG[2].Answer, out1 => "DB_STATUS_IJCORE".ANSWER_STA[2])
   END_RUNG
   RUNG wire#powerrail
      Contact( "AlwaysTRUE" )
   END_RUNG wire#w2
   RUNG wire#w2
      { S7_Templates := "SrcType := Int" } EQ_Contact(in1 := "DB_ProductionProgramActual".Program.MechanicalType, in2 := 0)
      Move(in := "DB_IJCoreMain".MSG[2].Answer, out1 => "DB_STATUS_IJCORE".ANSWER_STA[1])
   END_RUNG
   RUNG wire#powerrail
      Contact( "IJC_DB".MSG[3].DN )
      wire#w3
      Move(in := "DB_IJCoreMain".MSG[3].Answer, out1 => "DB_STATUS_IJCORE".ANSWER_STA[3])
   END_RUNG
   RUNG wire#powerrail
      Contact( "AlwaysTRUE" )
   END_RUNG wire#w3
   RUNG wire#powerrail
      Contact( "IJC_DB".MSG[4].DN )
      wire#w4
      Move(in := "DB_IJCoreMain".MSG[4].Answer, out1 => "DB_STATUS_IJCORE".ANSWER_STA[4])
   END_RUNG
   RUNG wire#powerrail
      Contact( "AlwaysTRUE" )
   END_RUNG wire#w4
   // the same network as SCL:
   #_w1 := "IJC_DB".MSG[1].DN OR "AlwaysTRUE";
   IF #_w1 AND ("DB_ProductionProgramActual".Program.MechanicalType = 1) THEN
       "DB_STATUS_IJCORE".ANSWER_STA[1] := "DB_IJCoreMain".MSG[1].Answer;
   END_IF;
   IF #_w1 AND ("DB_ProductionProgramActual".Program.MechanicalType = 0) THEN
       "DB_STATUS_IJCORE".ANSWER_STA[2] := "DB_IJCoreMain".MSG[1].Answer;
   END_IF;
   #_w2 := "IJC_DB".MSG[2].DN OR "AlwaysTRUE";
   IF #_w2 AND ("DB_ProductionProgramActual".Program.MechanicalType = 1) THEN
       "DB_STATUS_IJCORE".ANSWER_STA[2] := "DB_IJCoreMain".MSG[2].Answer;
   END_IF;
   IF #_w2 AND ("DB_ProductionProgramActual".Program.MechanicalType = 0) THEN
       "DB_STATUS_IJCORE".ANSWER_STA[1] := "DB_IJCoreMain".MSG[2].Answer;
   END_IF;
   IF "IJC_DB".MSG[3].DN OR "AlwaysTRUE" THEN
       "DB_STATUS_IJCORE".ANSWER_STA[3] := "DB_IJCoreMain".MSG[3].Answer;
   END_IF;
   IF "IJC_DB".MSG[4].DN OR "AlwaysTRUE" THEN
       "DB_STATUS_IJCORE".ANSWER_STA[4] := "DB_IJCoreMain".MSG[4].Answer;
   END_IF;
END_REGION

REGION Network 24: ANSWER TRC
   RUNG wire#powerrail
      Move(in := "DB_IJCoreMain".MSG[5].Answer, out1 => "DB_STATUS_IJCORE".ANSWER_TRC[1])
   END_RUNG
   RUNG wire#powerrail
      Move(in := "DB_IJCoreMain".MSG[6].Answer, out1 => "DB_STATUS_IJCORE".ANSWER_TRC[2])
   END_RUNG
   RUNG wire#powerrail
      Move(in := "DB_IJCoreMain".MSG[7].Answer, out1 => "DB_STATUS_IJCORE".ANSWER_TRC[3])
   END_RUNG
   RUNG wire#powerrail
      Move(in := "DB_IJCoreMain".MSG[8].Answer, out1 => "DB_STATUS_IJCORE".ANSWER_TRC[4])
   END_RUNG
   // the same network as SCL:
   "DB_STATUS_IJCORE".ANSWER_TRC[1] := "DB_IJCoreMain".MSG[5].Answer;
   "DB_STATUS_IJCORE".ANSWER_TRC[2] := "DB_IJCoreMain".MSG[6].Answer;
   "DB_STATUS_IJCORE".ANSWER_TRC[3] := "DB_IJCoreMain".MSG[7].Answer;
   "DB_STATUS_IJCORE".ANSWER_TRC[4] := "DB_IJCoreMain".MSG[8].Answer;
END_REGION

REGION Network 25: STATUS MSG TRC
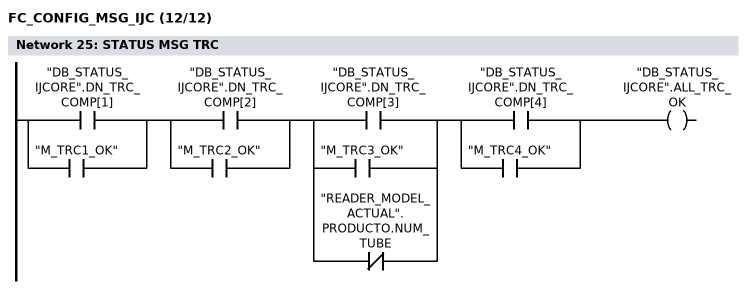
   RUNG wire#powerrail
      Contact( "DB_STATUS_IJCORE".DN_TRC_COMP[1] )
      wire#w1
      Contact( "DB_STATUS_IJCORE".DN_TRC_COMP[2] )
      wire#w2
      Contact( "DB_STATUS_IJCORE".DN_TRC_COMP[3] )
      wire#w3
      Contact( "DB_STATUS_IJCORE".DN_TRC_COMP[4] )
      wire#w4
      Coil( "DB_STATUS_IJCORE".ALL_TRC_OK )
   END_RUNG
   RUNG wire#powerrail
      Contact( "M_TRC1_OK" )
   END_RUNG wire#w1
   RUNG wire#w1
      Contact( "M_TRC2_OK" )
   END_RUNG wire#w2
   RUNG wire#w2
      Contact( "M_TRC3_OK" )
   END_RUNG wire#w3
   RUNG wire#w2
      I_Contact( "READER_MODEL_ACTUAL".PRODUCTO.NUM_TUBE )
   END_RUNG wire#w3
   RUNG wire#w3
      Contact( "M_TRC4_OK" )
   END_RUNG wire#w4
   // the same network as SCL:
   "DB_STATUS_IJCORE".ALL_TRC_OK := ("DB_STATUS_IJCORE".DN_TRC_COMP[1] OR "M_TRC1_OK") AND ("DB_STATUS_IJCORE".DN_TRC_COMP[2] OR "M_TRC2_OK") AND ("DB_STATUS_IJCORE".DN_TRC_COMP[3] OR "M_TRC3_OK" OR NOT "READER_MODEL_ACTUAL".PRODUCTO.NUM_TUBE) AND ("DB_STATUS_IJCORE".DN_TRC_COMP[4] OR "M_TRC4_OK");
END_REGION
END_FUNCTION
